LIN {X 0,Y 516.423,Z 190.622,A -85,B 0,C 180,E1 -4930.11,E2 -4930.11} C_VEL
LIN {X 0,Y 516.366,Z 194.851,A -85,B 0,C 180,E1 -4932.577,E2 -4932.577} C_VEL
LIN {X 0,Y 516.329,Z 197.599,A -85,B 0,C 180,E1 -4934.178,E2 -4934.178} C_VEL
LIN {X 0,Y 518.484,Z 209.749,A -85,B 0,C 180,E1 -4934.55,E2 -4934.55} C_VEL
LIN {X 0,Y 518.248,Z 221.683,A -85,B 0,C 180,E1 -4934.993,E2 -4934.993} C_VEL
LIN {X 0,Y 517.972,Z 233.125,A -85,B 0,C 180,E1 -4935.563,E2 -4935.563} C_VEL
LIN {X 0,Y 517.62,Z 243.966,A -85,B 0,C 180,E1 -4936.255,E2 -4936.255} C_VEL
LIN {X 0,Y 517.384,Z 254.996,A -85,B 0,C 180,E1 -4937.148,E2 -4937.148} C_VEL
LIN {X 0,Y 517.083,Z 264.736,A -85,B 0,C 180,E1 -4938.127,E2 -4938.127} C_VEL
LIN {X 0,Y 516.875,Z 273.613,A -85,B 0,C 180,E1 -4939.225,E2 -4939.225} C_VEL
LIN {X 0,Y 516.618,Z 281.309,A -85,B 0,C 180,E1 -4940.407,E2 -4940.407} C_VEL
LIN {X 0,Y 516.474,Z 288.372,A -85,B 0,C 180,E1 -4941.786,E2 -4941.786} C_VEL
LIN {X 0,Y 516.395,Z 293.063,A -85,B 0,C 180,E1 -4942.964,E2 -4942.964} C_VEL
LIN {X 0,Y 516.305,Z 296.646,A -85,B 0,C 180,E1 -4944.14,E2 -4944.14} C_VEL
LIN {X 0,Y 516.227,Z 299.218,A -85,B 0,C 180,E1 -4945.314,E2 -4945.314} C_VEL
LIN {X 0,Y 516.326,Z 300.425,A -85,B 0,C 180,E1 -4946.097,E2 -4946.097} C_VEL
LIN {X 0,Y 516.274,Z 301.209,A -85,B 0,C 180,E1 -4946.878,E2 -4946.878} C_VEL
LIN {X 0,Y 516.26,Z 301.586,A -85,B 0,C 180,E1 -4947.659,E2 -4947.659} C_VEL
LIN {X 0,Y 516.162,Z 301.206,A -85,B 0,C 180,E1 -4949.219,E2 -4949.219} C_VEL
LIN {X 0,Y 516.162,Z 300.418,A -85,B 0,C 180,E1 -4949.999,E2 -4949.999} C_VEL
LIN {X 0,Y 516.222,Z 297.602,A -85,B 0,C 180,E1 -4951.56,E2 -4951.56} C_VEL
LIN {X 0,Y 516.35,Z 294.377,A -85,B 0,C 180,E1 -4952.73,E2 -4952.73} C_VEL
LIN {X 0,Y 516.429,Z 290.102,A -85,B 0,C 180,E1 -4953.901,E2 -4953.901} C_VEL
LIN {X 0,Y 516.634,Z 284.648,A -85,B 0,C 180,E1 -4955.072,E2 -4955.072} C_VEL
LIN {X 0,Y 516.739,Z 277.853,A -85,B 0,C 180,E1 -4956.245,E2 -4956.245} C_VEL
LIN {X 0,Y 516.941,Z 269.359,A -85,B 0,C 180,E1 -4957.42,E2 -4957.42} C_VEL
LIN {X 0,Y 517.257,Z 260.641,A -85,B 0,C 180,E1 -4958.398,E2 -4958.398} C_VEL
LIN {X 0,Y 517.567,Z 249.918,A -85,B 0,C 180,E1 -4959.377,E2 -4959.377} C_VEL
LIN {X 0,Y 517.823,Z 239.153,A -85,B 0,C 180,E1 -4960.161,E2 -4960.161} C_VEL
LIN {X 0,Y 518.117,Z 227.088,A -85,B 0,C 180,E1 -4960.847,E2 -4960.847} C_VEL
LIN {X 0,Y 518.374,Z 215.239,A -85,B 0,C 180,E1 -4961.355,E2 -4961.355} C_VEL
LIN {X 0,Y 518.352,Z 208.104,A -85,B 0,C 180,E1 -4961.595,E2 -4961.595} C_VEL
LIN {X 0,Y 516.358,Z 197.517,A -85,B 0,C 180,E1 -4961.93,E2 -4961.93} C_VEL
LIN {X 0,Y 516.455,Z 192.31,A -85,B 0,C 180,E1 -4964.983,E2 -4964.983} C_VEL
LIN {X 0,Y 516.434,Z 186.816,A -85,B 0,C 180,E1 -4968.238,E2 -4968.238} C_VEL
LIN {X 0,Y 516.53,Z 182.754,A -85,B 0,C 180,E1 -4970.715,E2 -4970.715} C_VEL
LIN {X 0,Y 516.546,Z 178.687,A -85,B 0,C 180,E1 -4973.237,E2 -4973.237} C_VEL
LIN {X 0,Y 516.626,Z 174.098,A -85,B 0,C 180,E1 -4976.123,E2 -4976.123} C_VEL
LIN {X 0,Y 516.738,Z 169.128,A -85,B 0,C 180,E1 -4979.313,E2 -4979.313} C_VEL
LIN {X 0,Y 516.758,Z 164.99,A -85,B 0,C 180,E1 -4982.03,E2 -4982.03} C_VEL
LIN {X 0,Y 516.75,Z 163.594,A -85,B 0,C 180,E1 -4982.954,E2 -4982.954} C_VEL
LIN {X 0,Y 516.827,Z 163.108,A -85,B 0,C 180,E1 -4983.952,E2 -4983.952} C_VEL
LIN {X 0,Y 516.84,Z 163.107,A -85,B 0,C 180,E1 -4986.745,E2 -4986.745} C_VEL
LIN {X 0,Y 516.867,Z 163.102,A -85,B 0,C 180,E1 -4989.719,E2 -4989.719} C_VEL
LIN {X 0,Y 516.89,Z 163.097,A -85,B 0,C 180,E1 -4992.758,E2 -4992.758} C_VEL
LIN {X 0,Y 516.904,Z 163.097,A -85,B 0,C 180,E1 -4995.007,E2 -4995.007} C_VEL
LIN {X 0,Y 516.908,Z 163.094,A -85,B 0,C 180,E1 -4998.394,E2 -4998.394} C_VEL
LIN {X 0,Y 516.862,Z 163.101,A -85,B 0,C 180,E1 -5001.282,E2 -5001.282} C_VEL
LIN {X 0,Y 516.85,Z 163.106,A -85,B 0,C 180,E1 -5004.217,E2 -5004.217} C_VEL
LIN {X 0,Y 516.871,Z 163.101,A -85,B 0,C 180,E1 -5007.051,E2 -5007.051} C_VEL
LIN {X 0,Y 516.874,Z 163.101,A -85,B 0,C 180,E1 -5009.795,E2 -5009.795} C_VEL
LIN {X 0,Y 516.904,Z 163.097,A -85,B 0,C 180,E1 -5012.466,E2 -5012.466} C_VEL
LIN {X 0,Y 516.913,Z 163.095,A -85,B 0,C 180,E1 -5015.072,E2 -5015.072} C_VEL
LIN {X 0,Y 516.879,Z 163.099,A -85,B 0,C 180,E1 -5017.622,E2 -5017.622} C_VEL
LIN {X 0,Y 516.896,Z 163.1,A -85,B 0,C 180,E1 -5020.128,E2 -5020.128} C_VEL
LIN {X 0,Y 516.898,Z 163.097,A -85,B 0,C 180,E1 -5022.595,E2 -5022.595} C_VEL
LIN {X 0,Y 516.885,Z 163.098,A -85,B 0,C 180,E1 -5025.833,E2 -5025.833} C_VEL
LIN {X 0,Y 516.994,Z 163.087,A -85,B 0,C 180,E1 -5028.234,E2 -5028.234} C_VEL
LIN {X 0,Y 516.947,Z 163.089,A -85,B 0,C 180,E1 -5031.399,E2 -5031.399} C_VEL
LIN {X 0,Y 517.005,Z 163.087,A -85,B 0,C 180,E1 -5033.757,E2 -5033.757} C_VEL
LIN {X 0,Y 516.982,Z 163.087,A -85,B 0,C 180,E1 -5036.883,E2 -5036.883} C_VEL
LIN {X 0,Y 517.039,Z 163.079,A -85,B 0,C 180,E1 -5040,E2 -5040} C_VEL
LIN {X 0,Y 517.014,Z 163.083,A -85,B 0,C 180,E1 -5043.117,E2 -5043.117} C_VEL
LIN {X 0,Y 516.998,Z 163.086,A -85,B 0,C 180,E1 -5046.243,E2 -5046.243} C_VEL
LIN {X 0,Y 516.946,Z 163.089,A -85,B 0,C 180,E1 -5048.601,E2 -5048.601} C_VEL
LIN {X 0,Y 516.965,Z 163.088,A -85,B 0,C 180,E1 -5051.835,E2 -5051.835} C_VEL
LIN {X 0,Y 516.908,Z 163.097,A -85,B 0,C 180,E1 -5055.148,E2 -5055.148} C_VEL
LIN {X 0,Y 516.889,Z 163.101,A -85,B 0,C 180,E1 -5058.223,E2 -5058.223} C_VEL
LIN {X 0,Y 516.882,Z 163.099,A -85,B 0,C 180,E1 -5060.703,E2 -5060.703} C_VEL
LIN {X 0,Y 516.877,Z 163.103,A -85,B 0,C 180,E1 -5063.223,E2 -5063.223} C_VEL
LIN {X 0,Y 516.918,Z 163.093,A -85,B 0,C 180,E1 -5066.2,E2 -5066.2} C_VEL
LIN {X 0,Y 516.912,Z 163.094,A -85,B 0,C 180,E1 -5069.305,E2 -5069.305} C_VEL
LIN {X 0,Y 516.87,Z 163.102,A -85,B 0,C 180,E1 -5072.546,E2 -5072.546} C_VEL
LIN {X 0,Y 516.852,Z 163.105,A -85,B 0,C 180,E1 -5075.334,E2 -5075.334} C_VEL
LIN {X 0,Y 516.856,Z 163.103,A -85,B 0,C 180,E1 -5077.946,E2 -5077.946} C_VEL
LIN {X 0,Y 516.885,Z 163.103,A -85,B 0,C 180,E1 -5080.742,E2 -5080.742} C_VEL
LIN {X 0,Y 516.861,Z 163.101,A -85,B 0,C 180,E1 -5083.906,E2 -5083.906} C_VEL
LIN {X 0,Y 516.863,Z 163.106,A -85,B 0,C 180,E1 -5086.109,E2 -5086.109} C_VEL
LIN {X 0,Y 516.899,Z 163.1,A -85,B 0,C 180,E1 -5088.401,E2 -5088.401} C_VEL
LIN {X 0,Y 516.862,Z 163.107,A -85,B 0,C 180,E1 -5091.286,E2 -5091.286} C_VEL
LIN {X 0,Y 516.902,Z 163.236,A -85,B 0,C 180,E1 -5092.527,E2 -5092.527} C_VEL
LIN {X 0,Y 517.536,Z 167.733,A -85,B 0,C 180,E1 -5094.566,E2 -5094.566} C_VEL
LIN {X 0,Y 517.365,Z 174.379,A -85,B 0,C 180,E1 -5097.376,E2 -5097.376} C_VEL
LIN {X 0,Y 517.206,Z 181.852,A -85,B 0,C 180,E1 -5100.419,E2 -5100.419} C_VEL
LIN {X 0,Y 517,Z 190.448,A -85,B 0,C 180,E1 -5103.792,E2 -5103.792} C_VEL
LIN {X 0,Y 516.782,Z 198.275,A -85,B 0,C 180,E1 -5106.775,E2 -5106.775} C_VEL
LIN {X 0,Y 516.657,Z 206.41,A -85,B 0,C 180,E1 -5109.818,E2 -5109.818} C_VEL
LIN {X 0,Y 516.526,Z 213.919,A -85,B 0,C 180,E1 -5112.584,E2 -5112.584} C_VEL
LIN {X 0,Y 516.474,Z 221.738,A -85,B 0,C 180,E1 -5115.437,E2 -5115.437} C_VEL
LIN {X 0,Y 516.467,Z 223.583,A -85,B 0,C 180,E1 -5116.099,E2 -5116.099} C_VEL
LIN {X 0,Y 518.43,Z 237.052,A -85,B 0,C 180,E1 -5116.478,E2 -5116.478} C_VEL
LIN {X 0,Y 518.121,Z 250.37,A -85,B 0,C 180,E1 -5116.969,E2 -5116.969} C_VEL
LIN {X 0,Y 517.817,Z 263.139,A -85,B 0,C 180,E1 -5117.619,E2 -5117.619} C_VEL
LIN {X 0,Y 517.542,Z 274.076,A -85,B 0,C 180,E1 -5118.348,E2 -5118.348} C_VEL
LIN {X 0,Y 517.25,Z 284.743,A -85,B 0,C 180,E1 -5119.234,E2 -5119.234} C_VEL
LIN {X 0,Y 516.944,Z 294.354,A -85,B 0,C 180,E1 -5120.217,E2 -5120.217} C_VEL
LIN {X 0,Y 516.735,Z 302.234,A -85,B 0,C 180,E1 -5121.2,E2 -5121.2} C_VEL
LIN {X 0,Y 516.539,Z 309.929,A -85,B 0,C 180,E1 -5122.378,E2 -5122.378} C_VEL
LIN {X 0,Y 516.393,Z 317.023,A -85,B 0,C 180,E1 -5123.75,E2 -5123.75} C_VEL
LIN {X 0,Y 516.313,Z 321.743,A -85,B 0,C 180,E1 -5124.925,E2 -5124.925} C_VEL
LIN {X 0,Y 516.352,Z 325.351,A -85,B 0,C 180,E1 -5126.099,E2 -5126.099} C_VEL
LIN {X 0,Y 516.282,Z 327.209,A -85,B 0,C 180,E1 -5126.879,E2 -5126.879} C_VEL
LIN {X 0,Y 516.261,Z 328.603,A -85,B 0,C 180,E1 -5127.66,E2 -5127.66} C_VEL
LIN {X 0,Y 516.16,Z 330.203,A -85,B 0,C 180,E1 -5129.22,E2 -5129.22} C_VEL
LIN {X 0,Y 516.156,Z 330.418,A -85,B 0,C 180,E1 -5130.001,E2 -5130.001} C_VEL
LIN {X 0,Y 516.192,Z 329.596,A -85,B 0,C 180,E1 -5131.561,E2 -5131.561} C_VEL
LIN {X 0,Y 516.261,Z 328.603,A -85,B 0,C 180,E1 -5132.341,E2 -5132.341} C_VEL
LIN {X 0,Y 516.282,Z 327.209,A -85,B 0,C 180,E1 -5133.122,E2 -5133.122} C_VEL
LIN {X 0,Y 516.312,Z 324.275,A -85,B 0,C 180,E1 -5134.294,E2 -5134.294} C_VEL
LIN {X 0,Y 516.375,Z 320.304,A -85,B 0,C 180,E1 -5135.467,E2 -5135.467} C_VEL
LIN {X 0,Y 516.478,Z 314.404,A -85,B 0,C 180,E1 -5136.798,E2 -5136.798} C_VEL
LIN {X 0,Y 516.604,Z 307.521,A -85,B 0,C 180,E1 -5138.016,E2 -5138.016} C_VEL
LIN {X 0,Y 516.822,Z 299.24,A -85,B 0,C 180,E1 -5139.194,E2 -5139.194} C_VEL
LIN {X 0,Y 517.037,Z 290.752,A -85,B 0,C 180,E1 -5140.178,E2 -5140.178} C_VEL
LIN {X 0,Y 517.347,Z 280.265,A -85,B 0,C 180,E1 -5141.162,E2 -5141.162} C_VEL
LIN {X 0,Y 517.651,Z 269.287,A -85,B 0,C 180,E1 -5141.991,E2 -5141.991} C_VEL
LIN {X 0,Y 517.937,Z 258.519,A -85,B 0,C 180,E1 -5142.638,E2 -5142.638} C_VEL
LIN {X 0,Y 518.253,Z 246.86,A -85,B 0,C 180,E1 -5143.179,E2 -5143.179} C_VEL
LIN {X 0,Y 518.238,Z 235.249,A -85,B 0,C 180,E1 -5143.578,E2 -5143.578} C_VEL
LIN {X 0,Y 516.453,Z 223.564,A -85,B 0,C 180,E1 -5143.902,E2 -5143.902} C_VEL
LIN {X 0,Y 516.524,Z 214.964,A -85,B 0,C 180,E1 -5147.009,E2 -5147.009} C_VEL
LIN {X 0,Y 516.639,Z 207.215,A -85,B 0,C 180,E1 -5149.881,E2 -5149.881} C_VEL
LIN {X 0,Y 516.765,Z 199.392,A -85,B 0,C 180,E1 -5152.804,E2 -5152.804} C_VEL
LIN {X 0,Y 516.919,Z 192.705,A -85,B 0,C 180,E1 -5155.357,E2 -5155.357} C_VEL
LIN {X 0,Y 517.152,Z 184.948,A -85,B 0,C 180,E1 -5158.4,E2 -5158.4} C_VEL
LIN {X 0,Y 517.347,Z 177.234,A -85,B 0,C 180,E1 -5161.532,E2 -5161.532} C_VEL
LIN {X 0,Y 517.478,Z 171.26,A -85,B 0,C 180,E1 -5164.059,E2 -5164.059} C_VEL
LIN {X 0,Y 517.526,Z 167.439,A -85,B 0,C 180,E1 -5165.726,E2 -5165.726} C_VEL
LIN {X 0,Y 516.87,Z 163.106,A -85,B 0,C 180,E1 -5167.799,E2 -5167.799} C_VEL
LIN {X 0,Y 516.874,Z 163.101,A -85,B 0,C 180,E1 -5170.74,E2 -5170.74} C_VEL
LIN {X 0,Y 516.893,Z 163.097,A -85,B 0,C 180,E1 -5172.827,E2 -5172.827} C_VEL
LIN {X 0,Y 516.909,Z 163.099,A -85,B 0,C 180,E1 -5175.008,E2 -5175.008} C_VEL
LIN {X 0,Y 516.896,Z 163.1,A -85,B 0,C 180,E1 -5178.397,E2 -5178.397} C_VEL
LIN {X 0,Y 516.862,Z 163.102,A -85,B 0,C 180,E1 -5181.282,E2 -5181.282} C_VEL
LIN {X 0,Y 516.872,Z 163.099,A -85,B 0,C 180,E1 -5184.22,E2 -5184.22} C_VEL
LIN {X 0,Y 516.877,Z 163.104,A -85,B 0,C 180,E1 -5187.052,E2 -5187.052} C_VEL
LIN {X 0,Y 516.878,Z 163.1,A -85,B 0,C 180,E1 -5189.795,E2 -5189.795} C_VEL
LIN {X 0,Y 516.903,Z 163.098,A -85,B 0,C 180,E1 -5192.466,E2 -5192.466} C_VEL
LIN {X 0,Y 516.897,Z 163.099,A -85,B 0,C 180,E1 -5195.071,E2 -5195.071} C_VEL
LIN {X 0,Y 516.887,Z 163.097,A -85,B 0,C 180,E1 -5197.622,E2 -5197.622} C_VEL
LIN {X 0,Y 516.906,Z 163.097,A -85,B 0,C 180,E1 -5200.129,E2 -5200.129} C_VEL
LIN {X 0,Y 516.915,Z 163.097,A -85,B 0,C 180,E1 -5202.596,E2 -5202.596} C_VEL
LIN {X 0,Y 516.911,Z 163.097,A -85,B 0,C 180,E1 -5205.029,E2 -5205.029} C_VEL
LIN {X 0,Y 516.975,Z 163.087,A -85,B 0,C 180,E1 -5208.234,E2 -5208.234} C_VEL
LIN {X 0,Y 516.949,Z 163.089,A -85,B 0,C 180,E1 -5211.399,E2 -5211.399} C_VEL
LIN {X 0,Y 517.014,Z 163.084,A -85,B 0,C 180,E1 -5213.757,E2 -5213.757} C_VEL
LIN {X 0,Y 516.988,Z 163.088,A -85,B 0,C 180,E1 -5216.883,E2 -5216.883} C_VEL
LIN {X 0,Y 517.048,Z 163.078,A -85,B 0,C 180,E1 -5220,E2 -5220} C_VEL
LIN {X 0,Y 517.022,Z 163.08,A -85,B 0,C 180,E1 -5223.117,E2 -5223.117} C_VEL
LIN {X 0,Y 516.99,Z 163.086,A -85,B 0,C 180,E1 -5226.244,E2 -5226.244} C_VEL
LIN {X 0,Y 516.93,Z 163.096,A -85,B 0,C 180,E1 -5229.39,E2 -5229.39} C_VEL
LIN {X 0,Y 516.924,Z 163.094,A -85,B 0,C 180,E1 -5231.809,E2 -5231.809} C_VEL
LIN {X 0,Y 516.915,Z 163.094,A -85,B 0,C 180,E1 -5235.147,E2 -5235.147} C_VEL
LIN {X 0,Y 516.905,Z 163.095,A -85,B 0,C 180,E1 -5238.223,E2 -5238.223} C_VEL
LIN {X 0,Y 516.89,Z 163.1,A -85,B 0,C 180,E1 -5240.703,E2 -5240.703} C_VEL
LIN {X 0,Y 516.856,Z 163.103,A -85,B 0,C 180,E1 -5243.225,E2 -5243.225} C_VEL
LIN {X 0,Y 516.921,Z 163.096,A -85,B 0,C 180,E1 -5246.198,E2 -5246.198} C_VEL
LIN {X 0,Y 516.914,Z 163.1,A -85,B 0,C 180,E1 -5249.305,E2 -5249.305} C_VEL
LIN {X 0,Y 516.881,Z 163.102,A -85,B 0,C 180,E1 -5252.546,E2 -5252.546} C_VEL
LIN {X 0,Y 516.86,Z 163.102,A -85,B 0,C 180,E1 -5255.334,E2 -5255.334} C_VEL
LIN {X 0,Y 516.862,Z 163.104,A -85,B 0,C 180,E1 -5257.945,E2 -5257.945} C_VEL
LIN {X 0,Y 516.871,Z 163.102,A -85,B 0,C 180,E1 -5260.743,E2 -5260.743} C_VEL
LIN {X 0,Y 516.871,Z 163.104,A -85,B 0,C 180,E1 -5262.833,E2 -5262.833} C_VEL
LIN {X 0,Y 516.911,Z 163.095,A -85,B 0,C 180,E1 -5265.012,E2 -5265.012} C_VEL
LIN {X 0,Y 516.904,Z 163.097,A -85,B 0,C 180,E1 -5268.401,E2 -5268.401} C_VEL
LIN {X 0,Y 516.851,Z 163.103,A -85,B 0,C 180,E1 -5270.332,E2 -5270.332} C_VEL
LIN {X 0,Y 516.18,Z 163.195,A -85,B 0,C 180,E1 -5270.982,E2 -5270.982} C_VEL
LIN {X 0,Y 513.3,Z 163.735,A -85,B 0,C 180,E1 -5272.035,E2 -5272.035} C_VEL
LIN {X 0,Y 510.862,Z 164.526,A -85,B 0,C 180,E1 -5272.88,E2 -5272.88} C_VEL
LIN {X 0,Y 509.812,Z 165.338,A -85,B 0,C 180,E1 -5273.531,E2 -5273.531} C_VEL
LIN {X 0,Y 509.725,Z 165.651,A -85,B 0,C 180,E1 -5273.75,E2 -5273.75} C_VEL
LIN {X 0,Y 509.698,Z 169.763,A -85,B 0,C 180,E1 -5276.529,E2 -5276.529} C_VEL
LIN {X 0,Y 509.59,Z 173.994,A -85,B 0,C 180,E1 -5279.319,E2 -5279.319} C_VEL
LIN {X 0,Y 509.548,Z 178.187,A -85,B 0,C 180,E1 -5282.036,E2 -5282.036} C_VEL
LIN {X 0,Y 509.474,Z 182.359,A -85,B 0,C 180,E1 -5284.684,E2 -5284.684} C_VEL
LIN {X 0,Y 509.377,Z 187.013,A -85,B 0,C 180,E1 -5287.582,E2 -5287.582} C_VEL
LIN {X 0,Y 509.3,Z 192.127,A -85,B 0,C 180,E1 -5290.66,E2 -5290.66} C_VEL
LIN {X 0,Y 509.246,Z 196.339,A -85,B 0,C 180,E1 -5293.154,E2 -5293.154} C_VEL
LIN {X 0,Y 509.265,Z 197.751,A -85,B 0,C 180,E1 -5293.979,E2 -5293.979} C_VEL
LIN {X 0,Y 511.578,Z 210.681,A -85,B 0,C 180,E1 -5294.389,E2 -5294.389} C_VEL
LIN {X 0,Y 511.304,Z 222.986,A -85,B 0,C 180,E1 -5294.862,E2 -5294.862} C_VEL
LIN {X 0,Y 511.005,Z 234.608,A -85,B 0,C 180,E1 -5295.464,E2 -5295.464} C_VEL
LIN {X 0,Y 510.587,Z 246.462,A -85,B 0,C 180,E1 -5296.265,E2 -5296.265} C_VEL
LIN {X 0,Y 510.36,Z 257.042,A -85,B 0,C 180,E1 -5297.171,E2 -5297.171} C_VEL
LIN {X 0,Y 510.011,Z 266.994,A -85,B 0,C 180,E1 -5298.224,E2 -5298.224} C_VEL
LIN {X 0,Y 509.83,Z 275.011,A -85,B 0,C 180,E1 -5299.275,E2 -5299.275} C_VEL
LIN {X 0,Y 509.571,Z 282.468,A -85,B 0,C 180,E1 -5300.474,E2 -5300.474} C_VEL
LIN {X 0,Y 509.401,Z 288.446,A -85,B 0,C 180,E1 -5301.671,E2 -5301.671} C_VEL
LIN {X 0,Y 509.321,Z 293.164,A -85,B 0,C 180,E1 -5302.866,E2 -5302.866} C_VEL
LIN {X 0,Y 509.232,Z 296.77,A -85,B 0,C 180,E1 -5304.059,E2 -5304.059} C_VEL
LIN {X 0,Y 509.145,Z 299.366,A -85,B 0,C 180,E1 -5305.249,E2 -5305.249} C_VEL
LIN {X 0,Y 509.232,Z 300.585,A -85,B 0,C 180,E1 -5306.043,E2 -5306.043} C_VEL
LIN {X 0,Y 509.192,Z 301.39,A -85,B 0,C 180,E1 -5306.835,E2 -5306.835} C_VEL
LIN {X 0,Y 509.189,Z 301.778,A -85,B 0,C 180,E1 -5307.627,E2 -5307.627} C_VEL
LIN {X 0,Y 509.075,Z 301.42,A -85,B 0,C 180,E1 -5309.209,E2 -5309.209} C_VEL
LIN {X 0,Y 509.073,Z 300.653,A -85,B 0,C 180,E1 -5309.999,E2 -5309.999} C_VEL
LIN {X 0,Y 509.143,Z 297.86,A -85,B 0,C 180,E1 -5311.581,E2 -5311.581} C_VEL
LIN {X 0,Y 509.282,Z 294.659,A -85,B 0,C 180,E1 -5312.768,E2 -5312.768} C_VEL
LIN {X 0,Y 509.365,Z 290.409,A -85,B 0,C 180,E1 -5313.955,E2 -5313.955} C_VEL
LIN {X 0,Y 509.58,Z 284.983,A -85,B 0,C 180,E1 -5315.142,E2 -5315.142} C_VEL
LIN {X 0,Y 509.709,Z 278.218,A -85,B 0,C 180,E1 -5316.332,E2 -5316.332} C_VEL
LIN {X 0,Y 509.923,Z 269.779,A -85,B 0,C 180,E1 -5317.522,E2 -5317.522} C_VEL
LIN {X 0,Y 510.267,Z 261.104,A -85,B 0,C 180,E1 -5318.513,E2 -5318.513} C_VEL
LIN {X 0,Y 510.587,Z 250.436,A -85,B 0,C 180,E1 -5319.506,E2 -5319.506} C_VEL
LIN {X 0,Y 510.863,Z 239.78,A -85,B 0,C 180,E1 -5320.301,E2 -5320.301} C_VEL
LIN {X 0,Y 511.184,Z 227.828,A -85,B 0,C 180,E1 -5320.996,E2 -5320.996} C_VEL
LIN {X 0,Y 511.49,Z 215.533,A -85,B 0,C 180,E1 -5321.534,E2 -5321.534} C_VEL
LIN {X 0,Y 511.357,Z 208.331,A -85,B 0,C 180,E1 -5321.783,E2 -5321.783} C_VEL
LIN {X 0,Y 509.266,Z 197.718,A -85,B 0,C 180,E1 -5322.127,E2 -5322.127} C_VEL
LIN {X 0,Y 509.367,Z 192.502,A -85,B 0,C 180,E1 -5325.196,E2 -5325.196} C_VEL
LIN {X 0,Y 509.385,Z 188.102,A -85,B 0,C 180,E1 -5327.824,E2 -5327.824} C_VEL
LIN {X 0,Y 509.46,Z 182.923,A -85,B 0,C 180,E1 -5331.016,E2 -5331.016} C_VEL
LIN {X 0,Y 509.482,Z 178.842,A -85,B 0,C 180,E1 -5333.578,E2 -5333.578} C_VEL
LIN {X 0,Y 509.575,Z 174.566,A -85,B 0,C 180,E1 -5336.301,E2 -5336.301} C_VEL
LIN {X 0,Y 509.636,Z 170.633,A -85,B 0,C 180,E1 -5338.856,E2 -5338.856} C_VEL
LIN {X 0,Y 509.719,Z 166.487,A -85,B 0,C 180,E1 -5341.594,E2 -5341.594} C_VEL
LIN {X 0,Y 509.709,Z 163.998,A -85,B 0,C 180,E1 -5343.469,E2 -5343.469} C_VEL
LIN {X 0,Y 509.809,Z 163.98,A -85,B 0,C 180,E1 -5345.575,E2 -5345.575} C_VEL
LIN {X 0,Y 509.835,Z 163.979,A -85,B 0,C 180,E1 -5348.335,E2 -5348.335} C_VEL
LIN {X 0,Y 509.843,Z 163.976,A -85,B 0,C 180,E1 -5351.422,E2 -5351.422} C_VEL
LIN {X 0,Y 509.839,Z 163.975,A -85,B 0,C 180,E1 -5354.665,E2 -5354.665} C_VEL
LIN {X 0,Y 509.866,Z 163.971,A -85,B 0,C 180,E1 -5358.097,E2 -5358.097} C_VEL
LIN {X 0,Y 509.837,Z 163.98,A -85,B 0,C 180,E1 -5360.646,E2 -5360.646} C_VEL
LIN {X 0,Y 509.801,Z 163.982,A -85,B 0,C 180,E1 -5363.644,E2 -5363.644} C_VEL
LIN {X 0,Y 509.835,Z 163.977,A -85,B 0,C 180,E1 -5366.537,E2 -5366.537} C_VEL
LIN {X 0,Y 509.823,Z 163.982,A -85,B 0,C 180,E1 -5369.332,E2 -5369.332} C_VEL
LIN {X 0,Y 509.869,Z 163.971,A -85,B 0,C 180,E1 -5372.053,E2 -5372.053} C_VEL
LIN {X 0,Y 509.869,Z 163.976,A -85,B 0,C 180,E1 -5374.703,E2 -5374.703} C_VEL
LIN {X 0,Y 509.851,Z 163.974,A -85,B 0,C 180,E1 -5377.44,E2 -5377.44} C_VEL
LIN {X 0,Y 509.881,Z 163.974,A -85,B 0,C 180,E1 -5379.843,E2 -5379.843} C_VEL
LIN {X 0,Y 509.857,Z 163.977,A -85,B 0,C 180,E1 -5383.174,E2 -5383.174} C_VEL
LIN {X 0,Y 509.847,Z 163.976,A -85,B 0,C 180,E1 -5385.633,E2 -5385.633} C_VEL
LIN {X 0,Y 509.925,Z 163.967,A -85,B 0,C 180,E1 -5388.875,E2 -5388.875} C_VEL
LIN {X 0,Y 509.948,Z 163.968,A -85,B 0,C 180,E1 -5392.078,E2 -5392.078} C_VEL
LIN {X 0,Y 509.988,Z 163.957,A -85,B 0,C 180,E1 -5394.464,E2 -5394.464} C_VEL
LIN {X 0,Y 510.015,Z 163.957,A -85,B 0,C 180,E1 -5397.631,E2 -5397.631} C_VEL
LIN {X 0,Y 510.029,Z 163.955,A -85,B 0,C 180,E1 -5400.789,E2 -5400.789} C_VEL
LIN {X 0,Y 509.954,Z 163.962,A -85,B 0,C 180,E1 -5403.16,E2 -5403.16} C_VEL
LIN {X 0,Y 509.962,Z 163.962,A -85,B 0,C 180,E1 -5406.33,E2 -5406.33} C_VEL
LIN {X 0,Y 509.919,Z 163.964,A -85,B 0,C 180,E1 -5408.72,E2 -5408.72} C_VEL
LIN {X 0,Y 509.916,Z 163.965,A -85,B 0,C 180,E1 -5411.931,E2 -5411.931} C_VEL
LIN {X 0,Y 509.856,Z 163.975,A -85,B 0,C 180,E1 -5415.243,E2 -5415.243} C_VEL
LIN {X 0,Y 509.851,Z 163.978,A -85,B 0,C 180,E1 -5418.002,E2 -5418.002} C_VEL
LIN {X 0,Y 509.826,Z 163.978,A -85,B 0,C 180,E1 -5421.003,E2 -5421.003} C_VEL
LIN {X 0,Y 509.836,Z 163.979,A -85,B 0,C 180,E1 -5423.563,E2 -5423.563} C_VEL
LIN {X 0,Y 509.887,Z 163.969,A -85,B 0,C 180,E1 -5426.382,E2 -5426.382} C_VEL
LIN {X 0,Y 509.86,Z 163.977,A -85,B 0,C 180,E1 -5428.845,E2 -5428.845} C_VEL
LIN {X 0,Y 509.796,Z 163.982,A -85,B 0,C 180,E1 -5431.592,E2 -5431.592} C_VEL
LIN {X 0,Y 509.823,Z 163.979,A -85,B 0,C 180,E1 -5434.416,E2 -5434.416} C_VEL
LIN {X 0,Y 509.793,Z 163.985,A -85,B 0,C 180,E1 -5437.343,E2 -5437.343} C_VEL
LIN {X 0,Y 509.839,Z 163.977,A -85,B 0,C 180,E1 -5440.382,E2 -5440.382} C_VEL
LIN {X 0,Y 509.819,Z 163.979,A -85,B 0,C 180,E1 -5443.067,E2 -5443.067} C_VEL
LIN {X 0,Y 509.811,Z 163.981,A -85,B 0,C 180,E1 -5445.795,E2 -5445.795} C_VEL
LIN {X 0,Y 509.841,Z 163.979,A -85,B 0,C 180,E1 -5448.577,E2 -5448.577} C_VEL
LIN {X 0,Y 509.834,Z 163.981,A -85,B 0,C 180,E1 -5451.789,E2 -5451.789} C_VEL
LIN {X 0,Y 509.839,Z 164.11,A -85,B 0,C 180,E1 -5452.354,E2 -5452.354} C_VEL
LIN {X 0,Y 510.537,Z 169.183,A -85,B 0,C 180,E1 -5454.682,E2 -5454.682} C_VEL
LIN {X 0,Y 510.325,Z 175.809,A -85,B 0,C 180,E1 -5457.517,E2 -5457.517} C_VEL
LIN {X 0,Y 510.172,Z 183.589,A -85,B 0,C 180,E1 -5460.726,E2 -5460.726} C_VEL
LIN {X 0,Y 509.897,Z 192.538,A -85,B 0,C 180,E1 -5464.27,E2 -5464.27} C_VEL
LIN {X 0,Y 509.71,Z 200.377,A -85,B 0,C 180,E1 -5467.292,E2 -5467.292} C_VEL
LIN {X 0,Y 509.593,Z 207.09,A -85,B 0,C 180,E1 -5469.833,E2 -5469.833} C_VEL
LIN {X 0,Y 509.458,Z 214.878,A -85,B 0,C 180,E1 -5472.749,E2 -5472.749} C_VEL
LIN {X 0,Y 509.367,Z 223.383,A -85,B 0,C 180,E1 -5475.902,E2 -5475.902} C_VEL
LIN {X 0,Y 511.464,Z 237.235,A -85,B 0,C 180,E1 -5476.303,E2 -5476.303} C_VEL
LIN {X 0,Y 511.211,Z 250.172,A -85,B 0,C 180,E1 -5476.789,E2 -5476.789} C_VEL
LIN {X 0,Y 510.895,Z 261.567,A -85,B 0,C 180,E1 -5477.369,E2 -5477.369} C_VEL
LIN {X 0,Y 510.589,Z 272.564,A -85,B 0,C 180,E1 -5478.086,E2 -5478.086} C_VEL
LIN {X 0,Y 510.284,Z 283.472,A -85,B 0,C 180,E1 -5478.985,E2 -5478.985} C_VEL
LIN {X 0,Y 509.951,Z 292.367,A -85,B 0,C 180,E1 -5479.881,E2 -5479.881} C_VEL
LIN {X 0,Y 509.684,Z 302.035,A -85,B 0,C 180,E1 -5481.077,E2 -5481.077} C_VEL
LIN {X 0,Y 509.476,Z 309.731,A -85,B 0,C 180,E1 -5482.272,E2 -5482.272} C_VEL
LIN {X 0,Y 509.307,Z 316.825,A -85,B 0,C 180,E1 -5483.663,E2 -5483.663} C_VEL
LIN {X 0,Y 509.246,Z 321.546,A -85,B 0,C 180,E1 -5484.854,E2 -5484.854} C_VEL
LIN {X 0,Y 509.245,Z 325.153,A -85,B 0,C 180,E1 -5486.044,E2 -5486.044} C_VEL
LIN {X 0,Y 509.2,Z 327.012,A -85,B 0,C 180,E1 -5486.836,E2 -5486.836} C_VEL
LIN {X 0,Y 509.19,Z 328.406,A -85,B 0,C 180,E1 -5487.628,E2 -5487.628} C_VEL
LIN {X 0,Y 509.074,Z 330.005,A -85,B 0,C 180,E1 -5489.21,E2 -5489.21} C_VEL
LIN {X 0,Y 509.067,Z 330.221,A -85,B 0,C 180,E1 -5490.001,E2 -5490.001} C_VEL
LIN {X 0,Y 509.112,Z 329.399,A -85,B 0,C 180,E1 -5491.582,E2 -5491.582} C_VEL
LIN {X 0,Y 509.19,Z 328.406,A -85,B 0,C 180,E1 -5492.373,E2 -5492.373} C_VEL
LIN {X 0,Y 509.2,Z 327.011,A -85,B 0,C 180,E1 -5493.165,E2 -5493.165} C_VEL
LIN {X 0,Y 509.204,Z 324.076,A -85,B 0,C 180,E1 -5494.354,E2 -5494.354} C_VEL
LIN {X 0,Y 509.292,Z 320.105,A -85,B 0,C 180,E1 -5495.543,E2 -5495.543} C_VEL
LIN {X 0,Y 509.402,Z 314.452,A -85,B 0,C 180,E1 -5496.844,E2 -5496.844} C_VEL
LIN {X 0,Y 509.55,Z 307.322,A -85,B 0,C 180,E1 -5498.127,E2 -5498.127} C_VEL
LIN {X 0,Y 509.772,Z 299.04,A -85,B 0,C 180,E1 -5499.322,E2 -5499.322} C_VEL
LIN {X 0,Y 510.015,Z 290.552,A -85,B 0,C 180,E1 -5500.319,E2 -5500.319} C_VEL
LIN {X 0,Y 510.348,Z 280.065,A -85,B 0,C 180,E1 -5501.317,E2 -5501.317} C_VEL
LIN {X 0,Y 510.657,Z 269.087,A -85,B 0,C 180,E1 -5502.158,E2 -5502.158} C_VEL
LIN {X 0,Y 510.992,Z 258.319,A -85,B 0,C 180,E1 -5502.813,E2 -5502.813} C_VEL
LIN {X 0,Y 511.325,Z 246.66,A -85,B 0,C 180,E1 -5503.36,E2 -5503.36} C_VEL
LIN {X 0,Y 511.309,Z 235.964,A -85,B 0,C 180,E1 -5503.74,E2 -5503.74} C_VEL
LIN {X 0,Y 509.357,Z 223.36,A -85,B 0,C 180,E1 -5504.1,E2 -5504.1} C_VEL
LIN {X 0,Y 509.47,Z 214.833,A -85,B 0,C 180,E1 -5507.252,E2 -5507.252} C_VEL
LIN {X 0,Y 509.594,Z 206.71,A -85,B 0,C 180,E1 -5510.312,E2 -5510.312} C_VEL
LIN {X 0,Y 509.79,Z 198.171,A -85,B 0,C 180,E1 -5513.564,E2 -5513.564} C_VEL
LIN {X 0,Y 509.962,Z 190.945,A -85,B 0,C 180,E1 -5516.389,E2 -5516.389} C_VEL
LIN {X 0,Y 510.165,Z 183.775,A -85,B 0,C 180,E1 -5519.276,E2 -5519.276} C_VEL
LIN {X 0,Y 510.341,Z 177.187,A -85,B 0,C 180,E1 -5522.016,E2 -5522.016} C_VEL
LIN {X 0,Y 510.56,Z 170.658,A -85,B 0,C 180,E1 -5524.836,E2 -5524.836} C_VEL
LIN {X 0,Y 510.389,Z 167.421,A -85,B 0,C 180,E1 -5526.304,E2 -5526.304} C_VEL
LIN {X 0,Y 509.844,Z 163.983,A -85,B 0,C 180,E1 -5528.023,E2 -5528.023} C_VEL
LIN {X 0,Y 509.829,Z 163.979,A -85,B 0,C 180,E1 -5530.696,E2 -5530.696} C_VEL
LIN {X 0,Y 509.828,Z 163.978,A -85,B 0,C 180,E1 -5533.063,E2 -5533.063} C_VEL
LIN {X 0,Y 509.816,Z 163.98,A -85,B 0,C 180,E1 -5535.791,E2 -5535.791} C_VEL
LIN {X 0,Y 509.838,Z 163.979,A -85,B 0,C 180,E1 -5538.573,E2 -5538.573} C_VEL
LIN {X 0,Y 509.832,Z 163.981,A -85,B 0,C 180,E1 -5541.785,E2 -5541.785} C_VEL
LIN {X 0,Y 509.827,Z 163.976,A -85,B 0,C 180,E1 -5544.622,E2 -5544.622} C_VEL
LIN {X 0,Y 509.845,Z 163.976,A -85,B 0,C 180,E1 -5547.48,E2 -5547.48} C_VEL
LIN {X 0,Y 509.838,Z 163.979,A -85,B 0,C 180,E1 -5550.272,E2 -5550.272} C_VEL
LIN {X 0,Y 509.86,Z 163.974,A -85,B 0,C 180,E1 -5552.943,E2 -5552.943} C_VEL
LIN {X 0,Y 509.868,Z 163.975,A -85,B 0,C 180,E1 -5555.574,E2 -5555.574} C_VEL
LIN {X 0,Y 509.829,Z 163.976,A -85,B 0,C 180,E1 -5558.149,E2 -5558.149} C_VEL
LIN {X 0,Y 509.841,Z 163.98,A -85,B 0,C 180,E1 -5560.681,E2 -5560.681} C_VEL
LIN {X 0,Y 509.874,Z 163.972,A -85,B 0,C 180,E1 -5563.174,E2 -5563.174} C_VEL
LIN {X 0,Y 509.833,Z 163.979,A -85,B 0,C 180,E1 -5565.633,E2 -5565.633} C_VEL
LIN {X 0,Y 509.914,Z 163.971,A -85,B 0,C 180,E1 -5568.875,E2 -5568.875} C_VEL
LIN {X 0,Y 509.943,Z 163.965,A -85,B 0,C 180,E1 -5572.078,E2 -5572.078} C_VEL
LIN {X 0,Y 509.996,Z 163.958,A -85,B 0,C 180,E1 -5574.465,E2 -5574.465} C_VEL
LIN {X 0,Y 510.022,Z 163.956,A -85,B 0,C 180,E1 -5577.631,E2 -5577.631} C_VEL
LIN {X 0,Y 510.038,Z 163.954,A -85,B 0,C 180,E1 -5580.79,E2 -5580.79} C_VEL
LIN {X 0,Y 509.962,Z 163.959,A -85,B 0,C 180,E1 -5583.16,E2 -5583.16} C_VEL
LIN {X 0,Y 509.956,Z 163.962,A -85,B 0,C 180,E1 -5586.33,E2 -5586.33} C_VEL
LIN {X 0,Y 509.891,Z 163.972,A -85,B 0,C 180,E1 -5588.721,E2 -5588.721} C_VEL
LIN {X 0,Y 509.876,Z 163.973,A -85,B 0,C 180,E1 -5591.933,E2 -5591.933} C_VEL
LIN {X 0,Y 509.866,Z 163.972,A -85,B 0,C 180,E1 -5595.243,E2 -5595.243} C_VEL
LIN {X 0,Y 509.885,Z 163.971,A -85,B 0,C 180,E1 -5598.01,E2 -5598.01} C_VEL
LIN {X 0,Y 509.829,Z 163.981,A -85,B 0,C 180,E1 -5601.003,E2 -5601.003} C_VEL
LIN {X 0,Y 509.816,Z 163.98,A -85,B 0,C 180,E1 -5603.564,E2 -5603.564} C_VEL
LIN {X 0,Y 509.89,Z 163.971,A -85,B 0,C 180,E1 -5606.381,E2 -5606.381} C_VEL
LIN {X 0,Y 509.864,Z 163.973,A -85,B 0,C 180,E1 -5608.845,E2 -5608.845} C_VEL
LIN {X 0,Y 509.806,Z 163.98,A -85,B 0,C 180,E1 -5611.592,E2 -5611.592} C_VEL
LIN {X 0,Y 509.833,Z 163.98,A -85,B 0,C 180,E1 -5614.415,E2 -5614.415} C_VEL
LIN {X 0,Y 509.8,Z 163.984,A -85,B 0,C 180,E1 -5617.343,E2 -5617.343} C_VEL
LIN {X 0,Y 509.824,Z 163.978,A -85,B 0,C 180,E1 -5620.384,E2 -5620.384} C_VEL
LIN {X 0,Y 509.811,Z 163.981,A -85,B 0,C 180,E1 -5623.064,E2 -5623.064} C_VEL
LIN {X 0,Y 509.819,Z 163.98,A -85,B 0,C 180,E1 -5625.794,E2 -5625.794} C_VEL
LIN {X 0,Y 509.846,Z 163.976,A -85,B 0,C 180,E1 -5628.577,E2 -5628.577} C_VEL
LIN {X 0,Y 509.788,Z 163.984,A -85,B 0,C 180,E1 -5631.796,E2 -5631.796} C_VEL
LIN {X 0,Y 509.708,Z 164.057,A -85,B 0,C 180,E1 -5632.652,E2 -5632.652} C_VEL
LIN {X 0,Y 509.725,Z 165.651,A -85,B 0,C 180,E1 -5633.75,E2 -5633.75} C_VEL
LIN {X 0,Y 509.057,Z 166.693,A -85,B 0,C 180,E1 -5634.4,E2 -5634.4} C_VEL
LIN {X 0,Y 506.204,Z 168.582,A -85,B 0,C 180,E1 -5635.45,E2 -5635.45} C_VEL
LIN {X 0,Y 503.781,Z 170.119,A -85,B 0,C 180,E1 -5636.296,E2 -5636.296} C_VEL
LIN {X 0,Y 502.723,Z 171.212,A -85,B 0,C 180,E1 -5636.95,E2 -5636.95} C_VEL
LIN {X 0,Y 502.627,Z 171.554,A -85,B 0,C 180,E1 -5637.173,E2 -5637.173} C_VEL
LIN {X 0,Y 502.53,Z 175.999,A -85,B 0,C 180,E1 -5640.122,E2 -5640.122} C_VEL
LIN {X 0,Y 502.434,Z 179.669,A -85,B 0,C 180,E1 -5642.511,E2 -5642.511} C_VEL
LIN {X 0,Y 502.399,Z 184.186,A -85,B 0,C 180,E1 -5645.407,E2 -5645.407} C_VEL
LIN {X 0,Y 502.289,Z 188.011,A -85,B 0,C 180,E1 -5647.805,E2 -5647.805} C_VEL
LIN {X 0,Y 502.249,Z 192.247,A -85,B 0,C 180,E1 -5650.378,E2 -5650.378} C_VEL
LIN {X 0,Y 502.179,Z 196.453,A -85,B 0,C 180,E1 -5652.909,E2 -5652.909} C_VEL
LIN {X 0,Y 502.185,Z 197.891,A -85,B 0,C 180,E1 -5653.765,E2 -5653.765} C_VEL
LIN {X 0,Y 504.676,Z 211.346,A -85,B 0,C 180,E1 -5654.214,E2 -5654.214} C_VEL
LIN {X 0,Y 504.388,Z 223.694,A -85,B 0,C 180,E1 -5654.701,E2 -5654.701} C_VEL
LIN {X 0,Y 504.042,Z 236.006,A -85,B 0,C 180,E1 -5655.362,E2 -5655.362} C_VEL
LIN {X 0,Y 503.628,Z 247.599,A -85,B 0,C 180,E1 -5656.174,E2 -5656.174} C_VEL
LIN {X 0,Y 503.338,Z 258.016,A -85,B 0,C 180,E1 -5657.091,E2 -5657.091} C_VEL
LIN {X 0,Y 502.984,Z 267.64,A -85,B 0,C 180,E1 -5658.142,E2 -5658.142} C_VEL
LIN {X 0,Y 502.767,Z 276.376,A -85,B 0,C 180,E1 -5659.326,E2 -5659.326} C_VEL
LIN {X 0,Y 502.508,Z 283.627,A -85,B 0,C 180,E1 -5660.542,E2 -5660.542} C_VEL
LIN {X 0,Y 502.348,Z 288.519,A -85,B 0,C 180,E1 -5661.553,E2 -5661.553} C_VEL
LIN {X 0,Y 502.246,Z 293.264,A -85,B 0,C 180,E1 -5662.765,E2 -5662.765} C_VEL
LIN {X 0,Y 502.156,Z 296.458,A -85,B 0,C 180,E1 -5663.808,E2 -5663.808} C_VEL
LIN {X 0,Y 502.067,Z 299.514,A -85,B 0,C 180,E1 -5665.182,E2 -5665.182} C_VEL
LIN {X 0,Y 502.128,Z 300.744,A -85,B 0,C 180,E1 -5665.987,E2 -5665.987} C_VEL
LIN {X 0,Y 502.112,Z 301.57,A -85,B 0,C 180,E1 -5666.79,E2 -5666.79} C_VEL
LIN {X 0,Y 502.091,Z 301.97,A -85,B 0,C 180,E1 -5667.593,E2 -5667.593} C_VEL
LIN {X 0,Y 501.992,Z 301.633,A -85,B 0,C 180,E1 -5669.197,E2 -5669.197} C_VEL
LIN {X 0,Y 501.987,Z 300.885,A -85,B 0,C 180,E1 -5669.999,E2 -5669.999} C_VEL
LIN {X 0,Y 502.068,Z 298.118,A -85,B 0,C 180,E1 -5671.604,E2 -5671.604} C_VEL
LIN {X 0,Y 502.216,Z 294.94,A -85,B 0,C 180,E1 -5672.807,E2 -5672.807} C_VEL
LIN {X 0,Y 502.305,Z 290.716,A -85,B 0,C 180,E1 -5674.011,E2 -5674.011} C_VEL
LIN {X 0,Y 502.528,Z 285.318,A -85,B 0,C 180,E1 -5675.215,E2 -5675.215} C_VEL
LIN {X 0,Y 502.682,Z 278.583,A -85,B 0,C 180,E1 -5676.421,E2 -5676.421} C_VEL
LIN {X 0,Y 502.894,Z 270.2,A -85,B 0,C 180,E1 -5677.628,E2 -5677.628} C_VEL
LIN {X 0,Y 503.284,Z 261.567,A -85,B 0,C 180,E1 -5678.632,E2 -5678.632} C_VEL
LIN {X 0,Y 503.631,Z 250.953,A -85,B 0,C 180,E1 -5679.639,E2 -5679.639} C_VEL
LIN {X 0,Y 503.915,Z 240.389,A -85,B 0,C 180,E1 -5680.445,E2 -5680.445} C_VEL
LIN {X 0,Y 504.255,Z 228.568,A -85,B 0,C 180,E1 -5681.149,E2 -5681.149} C_VEL
LIN {X 0,Y 504.599,Z 215.511,A -85,B 0,C 180,E1 -5681.731,E2 -5681.731} C_VEL
LIN {X 0,Y 504.47,Z 209.425,A -85,B 0,C 180,E1 -5681.947,E2 -5681.947} C_VEL
LIN {X 0,Y 502.187,Z 197.88,A -85,B 0,C 180,E1 -5682.324,E2 -5682.324} C_VEL
LIN {X 0,Y 502.283,Z 192.704,A -85,B 0,C 180,E1 -5685.416,E2 -5685.416} C_VEL
LIN {X 0,Y 502.317,Z 188.528,A -85,B 0,C 180,E1 -5687.935,E2 -5687.935} C_VEL
LIN {X 0,Y 502.412,Z 184.451,A -85,B 0,C 180,E1 -5690.468,E2 -5690.468} C_VEL
LIN {X 0,Y 502.412,Z 180.362,A -85,B 0,C 180,E1 -5693.057,E2 -5693.057} C_VEL
LIN {X 0,Y 502.471,Z 176.261,A -85,B 0,C 180,E1 -5695.693,E2 -5695.693} C_VEL
LIN {X 0,Y 502.564,Z 172.136,A -85,B 0,C 180,E1 -5698.387,E2 -5698.387} C_VEL
LIN {X 0,Y 502.68,Z 167.985,A -85,B 0,C 180,E1 -5701.148,E2 -5701.148} C_VEL
LIN {X 0,Y 502.645,Z 165.203,A -85,B 0,C 180,E1 -5703.042,E2 -5703.042} C_VEL
LIN {X 0,Y 502.775,Z 164.86,A -85,B 0,C 180,E1 -5704.964,E2 -5704.964} C_VEL
LIN {X 0,Y 502.78,Z 164.858,A -85,B 0,C 180,E1 -5708.483,E2 -5708.483} C_VEL
LIN {X 0,Y 502.806,Z 164.852,A -85,B 0,C 180,E1 -5711.063,E2 -5711.063} C_VEL
LIN {X 0,Y 502.765,Z 164.86,A -85,B 0,C 180,E1 -5713.373,E2 -5713.373} C_VEL
LIN {X 0,Y 502.771,Z 164.858,A -85,B 0,C 180,E1 -5715.658,E2 -5715.658} C_VEL
LIN {X 0,Y 502.819,Z 164.849,A -85,B 0,C 180,E1 -5717.862,E2 -5717.862} C_VEL
LIN {X 0,Y 502.786,Z 164.857,A -85,B 0,C 180,E1 -5721.022,E2 -5721.022} C_VEL
LIN {X 0,Y 502.752,Z 164.862,A -85,B 0,C 180,E1 -5724.166,E2 -5724.166} C_VEL
LIN {X 0,Y 502.806,Z 164.853,A -85,B 0,C 180,E1 -5726.991,E2 -5726.991} C_VEL
LIN {X 0,Y 502.802,Z 164.853,A -85,B 0,C 180,E1 -5730.059,E2 -5730.059} C_VEL
LIN {X 0,Y 502.809,Z 164.853,A -85,B 0,C 180,E1 -5732.531,E2 -5732.531} C_VEL
LIN {X 0,Y 502.813,Z 164.85,A -85,B 0,C 180,E1 -5735.292,E2 -5735.292} C_VEL
LIN {X 0,Y 502.788,Z 164.855,A -85,B 0,C 180,E1 -5737.826,E2 -5737.826} C_VEL
LIN {X 0,Y 502.789,Z 164.855,A -85,B 0,C 180,E1 -5740.398,E2 -5740.398} C_VEL
LIN {X 0,Y 502.805,Z 164.854,A -85,B 0,C 180,E1 -5742.93,E2 -5742.93} C_VEL
LIN {X 0,Y 502.822,Z 164.853,A -85,B 0,C 180,E1 -5745.428,E2 -5745.428} C_VEL
LIN {X 0,Y 502.89,Z 164.844,A -85,B 0,C 180,E1 -5748.717,E2 -5748.717} C_VEL
LIN {X 0,Y 502.907,Z 164.843,A -85,B 0,C 180,E1 -5751.967,E2 -5751.967} C_VEL
LIN {X 0,Y 502.94,Z 164.835,A -85,B 0,C 180,E1 -5754.386,E2 -5754.386} C_VEL
LIN {X 0,Y 502.985,Z 164.833,A -85,B 0,C 180,E1 -5757.597,E2 -5757.597} C_VEL
LIN {X 0,Y 502.982,Z 164.83,A -85,B 0,C 180,E1 -5760,E2 -5760} C_VEL
LIN {X 0,Y 502.992,Z 164.832,A -85,B 0,C 180,E1 -5762.402,E2 -5762.402} C_VEL
LIN {X 0,Y 502.939,Z 164.837,A -85,B 0,C 180,E1 -5765.613,E2 -5765.613} C_VEL
LIN {X 0,Y 502.907,Z 164.841,A -85,B 0,C 180,E1 -5768.033,E2 -5768.033} C_VEL
LIN {X 0,Y 502.875,Z 164.849,A -85,B 0,C 180,E1 -5771.283,E2 -5771.283} C_VEL
LIN {X 0,Y 502.816,Z 164.853,A -85,B 0,C 180,E1 -5774.572,E2 -5774.572} C_VEL
LIN {X 0,Y 502.825,Z 164.853,A -85,B 0,C 180,E1 -5777.908,E2 -5777.908} C_VEL
LIN {X 0,Y 502.796,Z 164.854,A -85,B 0,C 180,E1 -5780.538,E2 -5780.538} C_VEL
LIN {X 0,Y 502.789,Z 164.856,A -85,B 0,C 180,E1 -5783.041,E2 -5783.041} C_VEL
LIN {X 0,Y 502.823,Z 164.85,A -85,B 0,C 180,E1 -5785.676,E2 -5785.676} C_VEL
LIN {X 0,Y 502.813,Z 164.852,A -85,B 0,C 180,E1 -5788.374,E2 -5788.374} C_VEL
LIN {X 0,Y 502.767,Z 164.857,A -85,B 0,C 180,E1 -5791.502,E2 -5791.502} C_VEL
LIN {X 0,Y 502.776,Z 164.857,A -85,B 0,C 180,E1 -5794.446,E2 -5794.446} C_VEL
LIN {X 0,Y 502.754,Z 164.862,A -85,B 0,C 180,E1 -5797.181,E2 -5797.181} C_VEL
LIN {X 0,Y 502.803,Z 164.852,A -85,B 0,C 180,E1 -5800.014,E2 -5800.014} C_VEL
LIN {X 0,Y 502.804,Z 164.853,A -85,B 0,C 180,E1 -5802.205,E2 -5802.205} C_VEL
LIN {X 0,Y 502.78,Z 164.854,A -85,B 0,C 180,E1 -5805.471,E2 -5805.471} C_VEL
LIN {X 0,Y 502.815,Z 164.857,A -85,B 0,C 180,E1 -5807.867,E2 -5807.867} C_VEL
LIN {X 0,Y 502.784,Z 164.86,A -85,B 0,C 180,E1 -5811.026,E2 -5811.026} C_VEL
LIN {X 0,Y 502.785,Z 164.925,A -85,B 0,C 180,E1 -5812.149,E2 -5812.149} C_VEL
LIN {X 0,Y 503.538,Z 170.193,A -85,B 0,C 180,E1 -5814.608,E2 -5814.608} C_VEL
LIN {X 0,Y 503.305,Z 176.814,A -85,B 0,C 180,E1 -5817.483,E2 -5817.483} C_VEL
LIN {X 0,Y 503.142,Z 184.58,A -85,B 0,C 180,E1 -5820.735,E2 -5820.735} C_VEL
LIN {X 0,Y 502.856,Z 193.52,A -85,B 0,C 180,E1 -5824.328,E2 -5824.328} C_VEL
LIN {X 0,Y 502.658,Z 201.216,A -85,B 0,C 180,E1 -5827.338,E2 -5827.338} C_VEL
LIN {X 0,Y 502.49,Z 209.161,A -85,B 0,C 180,E1 -5830.389,E2 -5830.389} C_VEL
LIN {X 0,Y 502.372,Z 216.947,A -85,B 0,C 180,E1 -5833.336,E2 -5833.336} C_VEL
LIN {X 0,Y 502.299,Z 223.229,A -85,B 0,C 180,E1 -5835.699,E2 -5835.699} C_VEL
LIN {X 0,Y 504.465,Z 237.417,A -85,B 0,C 180,E1 -5836.122,E2 -5836.122} C_VEL
LIN {X 0,Y 504.301,Z 249.975,A -85,B 0,C 180,E1 -5836.605,E2 -5836.605} C_VEL
LIN {X 0,Y 503.956,Z 261.517,A -85,B 0,C 180,E1 -5837.201,E2 -5837.201} C_VEL
LIN {X 0,Y 503.603,Z 272.365,A -85,B 0,C 180,E1 -5837.918,E2 -5837.918} C_VEL
LIN {X 0,Y 503.278,Z 283.274,A -85,B 0,C 180,E1 -5838.829,E2 -5838.829} C_VEL
LIN {X 0,Y 502.935,Z 292.169,A -85,B 0,C 180,E1 -5839.738,E2 -5839.738} C_VEL
LIN {X 0,Y 502.65,Z 301.837,A -85,B 0,C 180,E1 -5840.951,E2 -5840.951} C_VEL
LIN {X 0,Y 502.4,Z 309.532,A -85,B 0,C 180,E1 -5842.162,E2 -5842.162} C_VEL
LIN {X 0,Y 502.234,Z 316.627,A -85,B 0,C 180,E1 -5843.573,E2 -5843.573} C_VEL
LIN {X 0,Y 502.179,Z 321.348,A -85,B 0,C 180,E1 -5844.782,E2 -5844.782} C_VEL
LIN {X 0,Y 502.138,Z 324.954,A -85,B 0,C 180,E1 -5845.988,E2 -5845.988} C_VEL
LIN {X 0,Y 502.12,Z 326.814,A -85,B 0,C 180,E1 -5846.791,E2 -5846.791} C_VEL
LIN {X 0,Y 502.091,Z 328.208,A -85,B 0,C 180,E1 -5847.594,E2 -5847.594} C_VEL
LIN {X 0,Y 501.991,Z 329.808,A -85,B 0,C 180,E1 -5849.198,E2 -5849.198} C_VEL
LIN {X 0,Y 501.982,Z 330.024,A -85,B 0,C 180,E1 -5850.001,E2 -5850.001} C_VEL
LIN {X 0,Y 502.036,Z 329.201,A -85,B 0,C 180,E1 -5851.605,E2 -5851.605} C_VEL
LIN {X 0,Y 502.092,Z 328.208,A -85,B 0,C 180,E1 -5852.407,E2 -5852.407} C_VEL
LIN {X 0,Y 502.12,Z 326.813,A -85,B 0,C 180,E1 -5853.21,E2 -5853.21} C_VEL
LIN {X 0,Y 502.102,Z 323.877,A -85,B 0,C 180,E1 -5854.415,E2 -5854.415} C_VEL
LIN {X 0,Y 502.208,Z 319.907,A -85,B 0,C 180,E1 -5855.622,E2 -5855.622} C_VEL
LIN {X 0,Y 502.332,Z 313.9,A -85,B 0,C 180,E1 -5857.012,E2 -5857.012} C_VEL
LIN {X 0,Y 502.481,Z 307.122,A -85,B 0,C 180,E1 -5858.242,E2 -5858.242} C_VEL
LIN {X 0,Y 502.734,Z 298.84,A -85,B 0,C 180,E1 -5859.454,E2 -5859.454} C_VEL
LIN {X 0,Y 502.995,Z 290.352,A -85,B 0,C 180,E1 -5860.465,E2 -5860.465} C_VEL
LIN {X 0,Y 503.368,Z 279.866,A -85,B 0,C 180,E1 -5861.476,E2 -5861.476} C_VEL
LIN {X 0,Y 503.675,Z 268.887,A -85,B 0,C 180,E1 -5862.329,E2 -5862.329} C_VEL
LIN {X 0,Y 504.037,Z 258.12,A -85,B 0,C 180,E1 -5862.993,E2 -5862.993} C_VEL
LIN {X 0,Y 504.408,Z 246.461,A -85,B 0,C 180,E1 -5863.547,E2 -5863.547} C_VEL
LIN {X 0,Y 504.407,Z 236.983,A -85,B 0,C 180,E1 -5863.894,E2 -5863.894} C_VEL
LIN {X 0,Y 502.398,Z 224.229,A -85,B 0,C 180,E1 -5864.273,E2 -5864.273} C_VEL
LIN {X 0,Y 502.294,Z 223.129,A -85,B 0,C 180,E1 -5864.328,E2 -5864.328} C_VEL
LIN {X 0,Y 502.399,Z 214.69,A -85,B 0,C 180,E1 -5867.503,E2 -5867.503} C_VEL
LIN {X 0,Y 502.544,Z 206.971,A -85,B 0,C 180,E1 -5870.463,E2 -5870.463} C_VEL
LIN {X 0,Y 502.716,Z 199.176,A -85,B 0,C 180,E1 -5873.479,E2 -5873.479} C_VEL
LIN {X 0,Y 502.914,Z 191.388,A -85,B 0,C 180,E1 -5876.572,E2 -5876.572} C_VEL
LIN {X 0,Y 503.137,Z 184.806,A -85,B 0,C 180,E1 -5879.266,E2 -5879.266} C_VEL
LIN {X 0,Y 503.333,Z 178.239,A -85,B 0,C 180,E1 -5882.043,E2 -5882.043} C_VEL
LIN {X 0,Y 503.555,Z 171.707,A -85,B 0,C 180,E1 -5884.903,E2 -5884.903} C_VEL
LIN {X 0,Y 503.241,Z 167.403,A -85,B 0,C 180,E1 -5886.904,E2 -5886.904} C_VEL
LIN {X 0,Y 502.808,Z 164.859,A -85,B 0,C 180,E1 -5888.216,E2 -5888.216} C_VEL
LIN {X 0,Y 502.809,Z 164.852,A -85,B 0,C 180,E1 -5891.064,E2 -5891.064} C_VEL
LIN {X 0,Y 502.77,Z 164.859,A -85,B 0,C 180,E1 -5893.374,E2 -5893.374} C_VEL
LIN {X 0,Y 502.775,Z 164.858,A -85,B 0,C 180,E1 -5895.659,E2 -5895.659} C_VEL
LIN {X 0,Y 502.801,Z 164.855,A -85,B 0,C 180,E1 -5899.003,E2 -5899.003} C_VEL
LIN {X 0,Y 502.775,Z 164.859,A -85,B 0,C 180,E1 -5902.044,E2 -5902.044} C_VEL
LIN {X 0,Y 502.791,Z 164.855,A -85,B 0,C 180,E1 -5905.033,E2 -5905.033} C_VEL
LIN {X 0,Y 502.767,Z 164.857,A -85,B 0,C 180,E1 -5907.914,E2 -5907.914} C_VEL
LIN {X 0,Y 502.804,Z 164.856,A -85,B 0,C 180,E1 -5910.711,E2 -5910.711} C_VEL
LIN {X 0,Y 502.839,Z 164.851,A -85,B 0,C 180,E1 -5913.438,E2 -5913.438} C_VEL
LIN {X 0,Y 502.793,Z 164.853,A -85,B 0,C 180,E1 -5916.086,E2 -5916.086} C_VEL
LIN {X 0,Y 502.776,Z 164.859,A -85,B 0,C 180,E1 -5918.689,E2 -5918.689} C_VEL
LIN {X 0,Y 502.837,Z 164.85,A -85,B 0,C 180,E1 -5921.87,E2 -5921.87} C_VEL
LIN {X 0,Y 502.812,Z 164.852,A -85,B 0,C 180,E1 -5924.661,E2 -5924.661} C_VEL
LIN {X 0,Y 502.874,Z 164.844,A -85,B 0,C 180,E1 -5928.024,E2 -5928.024} C_VEL
LIN {X 0,Y 502.874,Z 164.843,A -85,B 0,C 180,E1 -5931.157,E2 -5931.157} C_VEL
LIN {X 0,Y 502.934,Z 164.837,A -85,B 0,C 180,E1 -5933.582,E2 -5933.582} C_VEL
LIN {X 0,Y 502.874,Z 164.845,A -85,B 0,C 180,E1 -5936.796,E2 -5936.796} C_VEL
LIN {X 0,Y 503.003,Z 164.83,A -85,B 0,C 180,E1 -5939.2,E2 -5939.2} C_VEL
LIN {X 0,Y 502.873,Z 164.843,A -85,B 0,C 180,E1 -5941.602,E2 -5941.602} C_VEL
LIN {X 0,Y 502.904,Z 164.838,A -85,B 0,C 180,E1 -5943.205,E2 -5943.205} C_VEL
LIN {X 0,Y 502.905,Z 164.84,A -85,B 0,C 180,E1 -5946.419,E2 -5946.419} C_VEL
LIN {X 0,Y 502.849,Z 164.849,A -85,B 0,C 180,E1 -5948.844,E2 -5948.844} C_VEL
LIN {X 0,Y 502.818,Z 164.854,A -85,B 0,C 180,E1 -5952.103,E2 -5952.103} C_VEL
LIN {X 0,Y 502.822,Z 164.851,A -85,B 0,C 180,E1 -5955.401,E2 -5955.401} C_VEL
LIN {X 0,Y 502.838,Z 164.848,A -85,B 0,C 180,E1 -5958.13,E2 -5958.13} C_VEL
LIN {X 0,Y 502.768,Z 164.859,A -85,B 0,C 180,E1 -5961.312,E2 -5961.312} C_VEL
LIN {X 0,Y 502.77,Z 164.86,A -85,B 0,C 180,E1 -5963.915,E2 -5963.915} C_VEL
LIN {X 0,Y 502.842,Z 164.848,A -85,B 0,C 180,E1 -5966.568,E2 -5966.568} C_VEL
LIN {X 0,Y 502.818,Z 164.856,A -85,B 0,C 180,E1 -5969.289,E2 -5969.289} C_VEL
LIN {X 0,Y 502.768,Z 164.857,A -85,B 0,C 180,E1 -5972.086,E2 -5972.086} C_VEL
LIN {X 0,Y 502.789,Z 164.855,A -85,B 0,C 180,E1 -5974.967,E2 -5974.967} C_VEL
LIN {X 0,Y 502.776,Z 164.858,A -85,B 0,C 180,E1 -5977.956,E2 -5977.956} C_VEL
LIN {X 0,Y 502.806,Z 164.856,A -85,B 0,C 180,E1 -5981.068,E2 -5981.068} C_VEL
LIN {X 0,Y 502.789,Z 164.859,A -85,B 0,C 180,E1 -5984.534,E2 -5984.534} C_VEL
LIN {X 0,Y 502.785,Z 164.857,A -85,B 0,C 180,E1 -5987.863,E2 -5987.863} C_VEL
LIN {X 0,Y 502.769,Z 164.857,A -85,B 0,C 180,E1 -5990.249,E2 -5990.249} C_VEL
LIN {X 0,Y 502.725,Z 164.864,A -85,B 0,C 180,E1 -5992.043,E2 -5992.043} C_VEL
LIN {X 0,Y 502.664,Z 165.539,A -85,B 0,C 180,E1 -5993.046,E2 -5993.046} C_VEL
LIN {X 0,Y 502.651,Z 169.819,A -85,B 0,C 180,E1 -5995.996,E2 -5995.996} C_VEL
LIN {X 0,Y 502.627,Z 171.554,A -85,B 0,C 180,E1 -5997.173,E2 -5997.173} C_VEL
LIN {X 0,Y 501.931,Z 172.619,A -85,B 0,C 180,E1 -5997.83,E2 -5997.83} C_VEL
LIN {X 0,Y 499.043,Z 174.539,A -85,B 0,C 180,E1 -5998.894,E2 -5998.894} C_VEL
LIN {X 0,Y 496.606,Z 176.095,A -85,B 0,C 180,E1 -5999.75,E2 -5999.75} C_VEL
LIN {X 0,Y 495.546,Z 177.209,A -85,B 0,C 180,E1 -6000.413,E2 -6000.413} C_VEL
LIN {X 0,Y 495.453,Z 177.557,A -85,B 0,C 180,E1 -6000.639,E2 -6000.639} C_VEL
LIN {X 0,Y 495.356,Z 181.703,A -85,B 0,C 180,E1 -6003.36,E2 -6003.36} C_VEL
LIN {X 0,Y 495.306,Z 185.333,A -85,B 0,C 180,E1 -6005.703,E2 -6005.703} C_VEL
LIN {X 0,Y 495.193,Z 189.536,A -85,B 0,C 180,E1 -6008.347,E2 -6008.347} C_VEL
LIN {X 0,Y 495.159,Z 193.776,A -85,B 0,C 180,E1 -6010.948,E2 -6010.948} C_VEL
LIN {X 0,Y 495.119,Z 198.224,A -85,B 0,C 180,E1 -6013.57,E2 -6013.57} C_VEL
LIN {X 0,Y 497.683,Z 211.397,A -85,B 0,C 180,E1 -6014.008,E2 -6014.008} C_VEL
LIN {X 0,Y 497.477,Z 224.445,A -85,B 0,C 180,E1 -6014.535,E2 -6014.535} C_VEL
LIN {X 0,Y 497.165,Z 235.79,A -85,B 0,C 180,E1 -6015.155,E2 -6015.155} C_VEL
LIN {X 0,Y 496.675,Z 247.454,A -85,B 0,C 180,E1 -6015.977,E2 -6015.977} C_VEL
LIN {X 0,Y 496.387,Z 257.925,A -85,B 0,C 180,E1 -6016.907,E2 -6016.907} C_VEL
LIN {X 0,Y 496.035,Z 266.67,A -85,B 0,C 180,E1 -6017.857,E2 -6017.857} C_VEL
LIN {X 0,Y 495.789,Z 275.035,A -85,B 0,C 180,E1 -6018.968,E2 -6018.968} C_VEL
LIN {X 0,Y 495.441,Z 282.557,A -85,B 0,C 180,E1 -6020.199,E2 -6020.199} C_VEL
LIN {X 0,Y 495.31,Z 288.593,A -85,B 0,C 180,E1 -6021.432,E2 -6021.432} C_VEL
LIN {X 0,Y 495.171,Z 293.364,A -85,B 0,C 180,E1 -6022.661,E2 -6022.661} C_VEL
LIN {X 0,Y 495.128,Z 296.056,A -85,B 0,C 180,E1 -6023.52,E2 -6023.52} C_VEL
LIN {X 0,Y 495.076,Z 298.017,A -85,B 0,C 180,E1 -6024.297,E2 -6024.297} C_VEL
LIN {X 0,Y 495.025,Z 300.904,A -85,B 0,C 180,E1 -6025.929,E2 -6025.929} C_VEL
LIN {X 0,Y 495.034,Z 301.748,A -85,B 0,C 180,E1 -6026.744,E2 -6026.744} C_VEL
LIN {X 0,Y 494.963,Z 302.194,A -85,B 0,C 180,E1 -6028.372,E2 -6028.372} C_VEL
LIN {X 0,Y 494.905,Z 301.115,A -85,B 0,C 180,E1 -6029.999,E2 -6029.999} C_VEL
LIN {X 0,Y 494.92,Z 299.948,A -85,B 0,C 180,E1 -6030.813,E2 -6030.813} C_VEL
LIN {X 0,Y 494.993,Z 298.376,A -85,B 0,C 180,E1 -6031.627,E2 -6031.627} C_VEL
LIN {X 0,Y 495.153,Z 295.222,A -85,B 0,C 180,E1 -6032.847,E2 -6032.847} C_VEL
LIN {X 0,Y 495.248,Z 291.023,A -85,B 0,C 180,E1 -6034.068,E2 -6034.068} C_VEL
LIN {X 0,Y 495.434,Z 284.658,A -85,B 0,C 180,E1 -6035.494,E2 -6035.494} C_VEL
LIN {X 0,Y 495.657,Z 278.948,A -85,B 0,C 180,E1 -6036.512,E2 -6036.512} C_VEL
LIN {X 0,Y 495.87,Z 270.618,A -85,B 0,C 180,E1 -6037.737,E2 -6037.737} C_VEL
LIN {X 0,Y 496.298,Z 262.027,A -85,B 0,C 180,E1 -6038.755,E2 -6038.755} C_VEL
LIN {X 0,Y 496.668,Z 251.463,A -85,B 0,C 180,E1 -6039.775,E2 -6039.775} C_VEL
LIN {X 0,Y 496.954,Z 240.965,A -85,B 0,C 180,E1 -6040.593,E2 -6040.593} C_VEL
LIN {X 0,Y 497.329,Z 229.277,A -85,B 0,C 180,E1 -6041.306,E2 -6041.306} C_VEL
LIN {X 0,Y 497.695,Z 216.729,A -85,B 0,C 180,E1 -6041.881,E2 -6041.881} C_VEL
LIN {X 0,Y 497.596,Z 210.384,A -85,B 0,C 180,E1 -6042.114,E2 -6042.114} C_VEL
LIN {X 0,Y 495.128,Z 198.066,A -85,B 0,C 180,E1 -6042.526,E2 -6042.526} C_VEL
LIN {X 0,Y 495.197,Z 192.905,A -85,B 0,C 180,E1 -6045.642,E2 -6045.642} C_VEL
LIN {X 0,Y 495.237,Z 188.728,A -85,B 0,C 180,E1 -6048.19,E2 -6048.19} C_VEL
LIN {X 0,Y 495.33,Z 184.622,A -85,B 0,C 180,E1 -6050.774,E2 -6050.774} C_VEL
LIN {X 0,Y 495.339,Z 180.514,A -85,B 0,C 180,E1 -6053.405,E2 -6053.405} C_VEL
LIN {X 0,Y 495.423,Z 176.404,A -85,B 0,C 180,E1 -6056.086,E2 -6056.086} C_VEL
LIN {X 0,Y 495.525,Z 172.271,A -85,B 0,C 180,E1 -6058.828,E2 -6058.828} C_VEL
LIN {X 0,Y 495.657,Z 168.013,A -85,B 0,C 180,E1 -6061.706,E2 -6061.706} C_VEL
LIN {X 0,Y 495.601,Z 165.833,A -85,B 0,C 180,E1 -6063.209,E2 -6063.209} C_VEL
LIN {X 0,Y 495.73,Z 165.735,A -85,B 0,C 180,E1 -6065.536,E2 -6065.536} C_VEL
LIN {X 0,Y 495.748,Z 165.735,A -85,B 0,C 180,E1 -6068.765,E2 -6068.765} C_VEL
LIN {X 0,Y 495.762,Z 165.734,A -85,B 0,C 180,E1 -6071.776,E2 -6071.776} C_VEL
LIN {X 0,Y 495.731,Z 165.735,A -85,B 0,C 180,E1 -6075.137,E2 -6075.137} C_VEL
LIN {X 0,Y 495.765,Z 165.727,A -85,B 0,C 180,E1 -6078.219,E2 -6078.219} C_VEL
LIN {X 0,Y 495.745,Z 165.732,A -85,B 0,C 180,E1 -6081.228,E2 -6081.228} C_VEL
LIN {X 0,Y 495.725,Z 165.738,A -85,B 0,C 180,E1 -6084.46,E2 -6084.46} C_VEL
LIN {X 0,Y 495.742,Z 165.736,A -85,B 0,C 180,E1 -6087.403,E2 -6087.403} C_VEL
LIN {X 0,Y 495.754,Z 165.73,A -85,B 0,C 180,E1 -6090.252,E2 -6090.252} C_VEL
LIN {X 0,Y 495.804,Z 165.725,A -85,B 0,C 180,E1 -6093.246,E2 -6093.246} C_VEL
LIN {X 0,Y 495.745,Z 165.73,A -85,B 0,C 180,E1 -6095.724,E2 -6095.724} C_VEL
LIN {X 0,Y 495.733,Z 165.736,A -85,B 0,C 180,E1 -6098.37,E2 -6098.37} C_VEL
LIN {X 0,Y 495.749,Z 165.732,A -85,B 0,C 180,E1 -6100.97,E2 -6100.97} C_VEL
LIN {X 0,Y 495.749,Z 165.734,A -85,B 0,C 180,E1 -6103.529,E2 -6103.529} C_VEL
LIN {X 0,Y 495.776,Z 165.728,A -85,B 0,C 180,E1 -6106.055,E2 -6106.055} C_VEL
LIN {X 0,Y 495.863,Z 165.721,A -85,B 0,C 180,E1 -6108.555,E2 -6108.555} C_VEL
LIN {X 0,Y 495.868,Z 165.719,A -85,B 0,C 180,E1 -6111.852,E2 -6111.852} C_VEL
LIN {X 0,Y 495.895,Z 165.713,A -85,B 0,C 180,E1 -6114.306,E2 -6114.306} C_VEL
LIN {X 0,Y 495.955,Z 165.709,A -85,B 0,C 180,E1 -6117.563,E2 -6117.563} C_VEL
LIN {X 0,Y 495.954,Z 165.706,A -85,B 0,C 180,E1 -6120,E2 -6120} C_VEL
LIN {X 0,Y 495.962,Z 165.707,A -85,B 0,C 180,E1 -6122.436,E2 -6122.436} C_VEL
LIN {X 0,Y 495.893,Z 165.716,A -85,B 0,C 180,E1 -6125.693,E2 -6125.693} C_VEL
LIN {X 0,Y 495.867,Z 165.717,A -85,B 0,C 180,E1 -6128.148,E2 -6128.148} C_VEL
LIN {X 0,Y 495.845,Z 165.722,A -85,B 0,C 180,E1 -6131.445,E2 -6131.445} C_VEL
LIN {X 0,Y 495.759,Z 165.733,A -85,B 0,C 180,E1 -6134.784,E2 -6134.784} C_VEL
LIN {X 0,Y 495.751,Z 165.731,A -85,B 0,C 180,E1 -6137.32,E2 -6137.32} C_VEL
LIN {X 0,Y 495.742,Z 165.735,A -85,B 0,C 180,E1 -6139.891,E2 -6139.891} C_VEL
LIN {X 0,Y 495.757,Z 165.731,A -85,B 0,C 180,E1 -6142.871,E2 -6142.871} C_VEL
LIN {X 0,Y 495.775,Z 165.726,A -85,B 0,C 180,E1 -6146.069,E2 -6146.069} C_VEL
LIN {X 0,Y 495.752,Z 165.735,A -85,B 0,C 180,E1 -6148.816,E2 -6148.816} C_VEL
LIN {X 0,Y 495.729,Z 165.735,A -85,B 0,C 180,E1 -6151.728,E2 -6151.728} C_VEL
LIN {X 0,Y 495.746,Z 165.732,A -85,B 0,C 180,E1 -6154.697,E2 -6154.697} C_VEL
LIN {X 0,Y 495.707,Z 165.739,A -85,B 0,C 180,E1 -6157.564,E2 -6157.564} C_VEL
LIN {X 0,Y 495.77,Z 165.728,A -85,B 0,C 180,E1 -6160.054,E2 -6160.054} C_VEL
LIN {X 0,Y 495.742,Z 165.733,A -85,B 0,C 180,E1 -6162.881,E2 -6162.881} C_VEL
LIN {X 0,Y 495.717,Z 165.739,A -85,B 0,C 180,E1 -6166.002,E2 -6166.002} C_VEL
LIN {X 0,Y 495.747,Z 165.735,A -85,B 0,C 180,E1 -6168.708,E2 -6168.708} C_VEL
LIN {X 0,Y 495.782,Z 165.857,A -85,B 0,C 180,E1 -6171.997,E2 -6171.997} C_VEL
LIN {X 0,Y 496.517,Z 171.195,A -85,B 0,C 180,E1 -6174.529,E2 -6174.529} C_VEL
LIN {X 0,Y 496.371,Z 175.978,A -85,B 0,C 180,E1 -6176.654,E2 -6176.654} C_VEL
LIN {X 0,Y 496.173,Z 183.248,A -85,B 0,C 180,E1 -6179.772,E2 -6179.772} C_VEL
LIN {X 0,Y 495.876,Z 190.027,A -85,B 0,C 180,E1 -6182.576,E2 -6182.576} C_VEL
LIN {X 0,Y 495.746,Z 196.368,A -85,B 0,C 180,E1 -6185.136,E2 -6185.136} C_VEL
LIN {X 0,Y 495.554,Z 204.547,A -85,B 0,C 180,E1 -6188.365,E2 -6188.365} C_VEL
LIN {X 0,Y 495.383,Z 212.335,A -85,B 0,C 180,E1 -6191.387,E2 -6191.387} C_VEL
LIN {X 0,Y 495.242,Z 220.085,A -85,B 0,C 180,E1 -6194.36,E2 -6194.36} C_VEL
LIN {X 0,Y 495.212,Z 223.177,A -85,B 0,C 180,E1 -6195.503,E2 -6195.503} C_VEL
LIN {X 0,Y 497.251,Z 236.407,A -85,B 0,C 180,E1 -6195.89,E2 -6195.89} C_VEL
LIN {X 0,Y 497.608,Z 241.009,A -85,B 0,C 180,E1 -6196.057,E2 -6196.057} C_VEL
LIN {X 0,Y 497.228,Z 254.033,A -85,B 0,C 180,E1 -6196.619,E2 -6196.619} C_VEL
LIN {X 0,Y 496.809,Z 266.284,A -85,B 0,C 180,E1 -6197.332,E2 -6197.332} C_VEL
LIN {X 0,Y 496.515,Z 277.333,A -85,B 0,C 180,E1 -6198.158,E2 -6198.158} C_VEL
LIN {X 0,Y 496.19,Z 286.266,A -85,B 0,C 180,E1 -6198.978,E2 -6198.978} C_VEL
LIN {X 0,Y 495.796,Z 295.438,A -85,B 0,C 180,E1 -6200.001,E2 -6200.001} C_VEL
LIN {X 0,Y 495.519,Z 304.378,A -85,B 0,C 180,E1 -6201.231,E2 -6201.231} C_VEL
LIN {X 0,Y 495.277,Z 311.573,A -85,B 0,C 180,E1 -6202.459,E2 -6202.459} C_VEL
LIN {X 0,Y 495.123,Z 317.614,A -85,B 0,C 180,E1 -6203.761,E2 -6203.761} C_VEL
LIN {X 0,Y 495.036,Z 322.461,A -85,B 0,C 180,E1 -6205.114,E2 -6205.114} C_VEL
LIN {X 0,Y 495.031,Z 324.756,A -85,B 0,C 180,E1 -6205.93,E2 -6205.93} C_VEL
LIN {X 0,Y 495.041,Z 326.617,A -85,B 0,C 180,E1 -6206.745,E2 -6206.745} C_VEL
LIN {X 0,Y 494.998,Z 328.011,A -85,B 0,C 180,E1 -6207.56,E2 -6207.56} C_VEL
LIN {X 0,Y 494.962,Z 329.005,A -85,B 0,C 180,E1 -6208.373,E2 -6208.373} C_VEL
LIN {X 0,Y 494.899,Z 329.826,A -85,B 0,C 180,E1 -6210.001,E2 -6210.001} C_VEL
LIN {X 0,Y 494.962,Z 329.004,A -85,B 0,C 180,E1 -6211.628,E2 -6211.628} C_VEL
LIN {X 0,Y 494.998,Z 328.01,A -85,B 0,C 180,E1 -6212.442,E2 -6212.442} C_VEL
LIN {X 0,Y 495.042,Z 326.615,A -85,B 0,C 180,E1 -6213.256,E2 -6213.256} C_VEL
LIN {X 0,Y 495.007,Z 323.679,A -85,B 0,C 180,E1 -6214.479,E2 -6214.479} C_VEL
LIN {X 0,Y 495.125,Z 319.708,A -85,B 0,C 180,E1 -6215.702,E2 -6215.702} C_VEL
LIN {X 0,Y 495.256,Z 313.599,A -85,B 0,C 180,E1 -6217.133,E2 -6217.133} C_VEL
LIN {X 0,Y 495.428,Z 306.923,A -85,B 0,C 180,E1 -6218.361,E2 -6218.361} C_VEL
LIN {X 0,Y 495.704,Z 298.641,A -85,B 0,C 180,E1 -6219.589,E2 -6219.589} C_VEL
LIN {X 0,Y 495.989,Z 290.153,A -85,B 0,C 180,E1 -6220.615,E2 -6220.615} C_VEL
LIN {X 0,Y 496.385,Z 279.668,A -85,B 0,C 180,E1 -6221.639,E2 -6221.639} C_VEL
LIN {X 0,Y 496.743,Z 268.484,A -85,B 0,C 180,E1 -6222.519,E2 -6222.519} C_VEL
LIN {X 0,Y 497.091,Z 257.931,A -85,B 0,C 180,E1 -6223.178,E2 -6223.178} C_VEL
LIN {X 0,Y 497.501,Z 246.288,A -85,B 0,C 180,E1 -6223.739,E2 -6223.739} C_VEL
LIN {X 0,Y 497.459,Z 237.585,A -85,B 0,C 180,E1 -6224.066,E2 -6224.066} C_VEL
LIN {X 0,Y 495.335,Z 224.195,A -85,B 0,C 180,E1 -6224.481,E2 -6224.481} C_VEL
LIN {X 0,Y 495.189,Z 222.953,A -85,B 0,C 180,E1 -6224.538,E2 -6224.538} C_VEL
LIN {X 0,Y 495.324,Z 215.644,A -85,B 0,C 180,E1 -6227.335,E2 -6227.335} C_VEL
LIN {X 0,Y 495.48,Z 207.316,A -85,B 0,C 180,E1 -6230.584,E2 -6230.584} C_VEL
LIN {X 0,Y 495.691,Z 199.066,A -85,B 0,C 180,E1 -6233.832,E2 -6233.832} C_VEL
LIN {X 0,Y 495.864,Z 191.839,A -85,B 0,C 180,E1 -6236.758,E2 -6236.758} C_VEL
LIN {X 0,Y 496.138,Z 184.74,A -85,B 0,C 180,E1 -6239.72,E2 -6239.72} C_VEL
LIN {X 0,Y 496.366,Z 178.176,A -85,B 0,C 180,E1 -6242.548,E2 -6242.548} C_VEL
LIN {X 0,Y 496.575,Z 171.677,A -85,B 0,C 180,E1 -6245.467,E2 -6245.467} C_VEL
LIN {X 0,Y 495.86,Z 166.325,A -85,B 0,C 180,E1 -6248.061,E2 -6248.061} C_VEL
LIN {X 0,Y 495.77,Z 165.736,A -85,B 0,C 180,E1 -6248.457,E2 -6248.457} C_VEL
LIN {X 0,Y 495.766,Z 165.733,A -85,B 0,C 180,E1 -6251.777,E2 -6251.777} C_VEL
LIN {X 0,Y 495.735,Z 165.736,A -85,B 0,C 180,E1 -6255.138,E2 -6255.138} C_VEL
LIN {X 0,Y 495.74,Z 165.735,A -85,B 0,C 180,E1 -6258.217,E2 -6258.217} C_VEL
LIN {X 0,Y 495.732,Z 165.735,A -85,B 0,C 180,E1 -6261.407,E2 -6261.407} C_VEL
LIN {X 0,Y 495.739,Z 165.731,A -85,B 0,C 180,E1 -6264.462,E2 -6264.462} C_VEL
LIN {X 0,Y 495.749,Z 165.733,A -85,B 0,C 180,E1 -6267.404,E2 -6267.404} C_VEL
LIN {X 0,Y 495.746,Z 165.733,A -85,B 0,C 180,E1 -6270.252,E2 -6270.252} C_VEL
LIN {X 0,Y 495.8,Z 165.727,A -85,B 0,C 180,E1 -6273.249,E2 -6273.249} C_VEL
LIN {X 0,Y 495.746,Z 165.733,A -85,B 0,C 180,E1 -6275.725,E2 -6275.725} C_VEL
LIN {X 0,Y 495.741,Z 165.732,A -85,B 0,C 180,E1 -6278.371,E2 -6278.371} C_VEL
LIN {X 0,Y 495.805,Z 165.726,A -85,B 0,C 180,E1 -6281.743,E2 -6281.743} C_VEL
LIN {X 0,Y 495.796,Z 165.726,A -85,B 0,C 180,E1 -6284.547,E2 -6284.547} C_VEL
LIN {X 0,Y 495.851,Z 165.719,A -85,B 0,C 180,E1 -6287.937,E2 -6287.937} C_VEL
LIN {X 0,Y 495.837,Z 165.72,A -85,B 0,C 180,E1 -6291.03,E2 -6291.03} C_VEL
LIN {X 0,Y 495.886,Z 165.715,A -85,B 0,C 180,E1 -6293.49,E2 -6293.49} C_VEL
LIN {X 0,Y 495.819,Z 165.724,A -85,B 0,C 180,E1 -6296.75,E2 -6296.75} C_VEL
LIN {X 0,Y 495.953,Z 165.708,A -85,B 0,C 180,E1 -6299.188,E2 -6299.188} C_VEL
LIN {X 0,Y 495.842,Z 165.719,A -85,B 0,C 180,E1 -6301.625,E2 -6301.625} C_VEL
LIN {X 0,Y 495.848,Z 165.717,A -85,B 0,C 180,E1 -6303.25,E2 -6303.25} C_VEL
LIN {X 0,Y 495.856,Z 165.718,A -85,B 0,C 180,E1 -6306.511,E2 -6306.511} C_VEL
LIN {X 0,Y 495.817,Z 165.725,A -85,B 0,C 180,E1 -6308.97,E2 -6308.97} C_VEL
LIN {X 0,Y 495.8,Z 165.727,A -85,B 0,C 180,E1 -6312.036,E2 -6312.036} C_VEL
LIN {X 0,Y 495.798,Z 165.726,A -85,B 0,C 180,E1 -6315.453,E2 -6315.453} C_VEL
LIN {X 0,Y 495.806,Z 165.723,A -85,B 0,C 180,E1 -6318.257,E2 -6318.257} C_VEL
LIN {X 0,Y 495.732,Z 165.734,A -85,B 0,C 180,E1 -6321.63,E2 -6321.63} C_VEL
LIN {X 0,Y 495.756,Z 165.731,A -85,B 0,C 180,E1 -6324.875,E2 -6324.875} C_VEL
LIN {X 0,Y 495.792,Z 165.726,A -85,B 0,C 180,E1 -6326.976,E2 -6326.976} C_VEL
LIN {X 0,Y 495.756,Z 165.729,A -85,B 0,C 180,E1 -6330.151,E2 -6330.151} C_VEL
LIN {X 0,Y 495.775,Z 165.729,A -85,B 0,C 180,E1 -6333.246,E2 -6333.246} C_VEL
LIN {X 0,Y 495.708,Z 165.738,A -85,B 0,C 180,E1 -6336.091,E2 -6336.091} C_VEL
LIN {X 0,Y 495.747,Z 165.732,A -85,B 0,C 180,E1 -6338.77,E2 -6338.77} C_VEL
LIN {X 0,Y 495.744,Z 165.73,A -85,B 0,C 180,E1 -6341.783,E2 -6341.783} C_VEL
LIN {X 0,Y 495.738,Z 165.733,A -85,B 0,C 180,E1 -6345.141,E2 -6345.141} C_VEL
LIN {X 0,Y 495.746,Z 165.734,A -85,B 0,C 180,E1 -6348.221,E2 -6348.221} C_VEL
LIN {X 0,Y 495.724,Z 165.74,A -85,B 0,C 180,E1 -6351.238,E2 -6351.238} C_VEL
LIN {X 0,Y 495.613,Z 165.776,A -85,B 0,C 180,E1 -6352.571,E2 -6352.571} C_VEL
LIN {X 0,Y 495.619,Z 169.87,A -85,B 0,C 180,E1 -6355.446,E2 -6355.446} C_VEL
LIN {X 0,Y 495.542,Z 174.132,A -85,B 0,C 180,E1 -6358.35,E2 -6358.35} C_VEL
LIN {X 0,Y 495.453,Z 177.557,A -85,B 0,C 180,E1 -6360.639,E2 -6360.639} C_VEL
LIN {X 0,Y 494.752,Z 178.642,A -85,B 0,C 180,E1 -6361.305,E2 -6361.305} C_VEL
LIN {X 0,Y 491.838,Z 180.581,A -85,B 0,C 180,E1 -6362.383,E2 -6362.383} C_VEL
LIN {X 0,Y 489.389,Z 182.151,A -85,B 0,C 180,E1 -6363.251,E2 -6363.251} C_VEL
LIN {X 0,Y 488.342,Z 183.281,A -85,B 0,C 180,E1 -6363.924,E2 -6363.924} C_VEL
LIN {X 0,Y 488.258,Z 183.638,A -85,B 0,C 180,E1 -6364.152,E2 -6364.152} C_VEL
LIN {X 0,Y 488.212,Z 188.216,A -85,B 0,C 180,E1 -6367.119,E2 -6367.119} C_VEL
LIN {X 0,Y 488.104,Z 193.909,A -85,B 0,C 180,E1 -6370.661,E2 -6370.661} C_VEL
LIN {X 0,Y 488.024,Z 198.269,A -85,B 0,C 180,E1 -6373.335,E2 -6373.335} C_VEL
LIN {X 0,Y 490.869,Z 212.669,A -85,B 0,C 180,E1 -6373.842,E2 -6373.842} C_VEL
LIN {X 0,Y 490.601,Z 225.257,A -85,B 0,C 180,E1 -6374.366,E2 -6374.366} C_VEL
LIN {X 0,Y 490.179,Z 237.212,A -85,B 0,C 180,E1 -6375.045,E2 -6375.045} C_VEL
LIN {X 0,Y 489.706,Z 248.644,A -85,B 0,C 180,E1 -6375.879,E2 -6375.879} C_VEL
LIN {X 0,Y 489.389,Z 258.934,A -85,B 0,C 180,E1 -6376.822,E2 -6376.822} C_VEL
LIN {X 0,Y 488.942,Z 268.913,A -85,B 0,C 180,E1 -6377.964,E2 -6377.964} C_VEL
LIN {X 0,Y 488.698,Z 277.771,A -85,B 0,C 180,E1 -6379.225,E2 -6379.225} C_VEL
LIN {X 0,Y 488.388,Z 284.808,A -85,B 0,C 180,E1 -6380.475,E2 -6380.475} C_VEL
LIN {X 0,Y 488.193,Z 290.415,A -85,B 0,C 180,E1 -6381.723,E2 -6381.723} C_VEL
LIN {X 0,Y 488.073,Z 294.821,A -85,B 0,C 180,E1 -6382.97,E2 -6382.97} C_VEL
LIN {X 0,Y 488,Z 298.155,A -85,B 0,C 180,E1 -6384.214,E2 -6384.214} C_VEL
LIN {X 0,Y 487.924,Z 301.064,A -85,B 0,C 180,E1 -6385.87,E2 -6385.87} C_VEL
LIN {X 0,Y 487.957,Z 301.924,A -85,B 0,C 180,E1 -6386.697,E2 -6386.697} C_VEL
LIN {X 0,Y 487.891,Z 302.396,A -85,B 0,C 180,E1 -6388.349,E2 -6388.349} C_VEL
LIN {X 0,Y 487.825,Z 301.343,A -85,B 0,C 180,E1 -6389.999,E2 -6389.999} C_VEL
LIN {X 0,Y 487.843,Z 300.194,A -85,B 0,C 180,E1 -6390.825,E2 -6390.825} C_VEL
LIN {X 0,Y 487.922,Z 298.633,A -85,B 0,C 180,E1 -6391.65,E2 -6391.65} C_VEL
LIN {X 0,Y 488.091,Z 295.501,A -85,B 0,C 180,E1 -6392.888,E2 -6392.888} C_VEL
LIN {X 0,Y 488.193,Z 291.326,A -85,B 0,C 180,E1 -6394.127,E2 -6394.127} C_VEL
LIN {X 0,Y 488.373,Z 284.985,A -85,B 0,C 180,E1 -6395.573,E2 -6395.573} C_VEL
LIN {X 0,Y 488.696,Z 277.913,A -85,B 0,C 180,E1 -6396.836,E2 -6396.836} C_VEL
LIN {X 0,Y 488.927,Z 269.4,A -85,B 0,C 180,E1 -6398.055,E2 -6398.055} C_VEL
LIN {X 0,Y 489.345,Z 260.525,A -85,B 0,C 180,E1 -6399.089,E2 -6399.089} C_VEL
LIN {X 0,Y 489.75,Z 250.77,A -85,B 0,C 180,E1 -6400.019,E2 -6400.019} C_VEL
LIN {X 0,Y 490.084,Z 240.015,A -85,B 0,C 180,E1 -6400.847,E2 -6400.847} C_VEL
LIN {X 0,Y 490.433,Z 227.955,A -85,B 0,C 180,E1 -6401.572,E2 -6401.572} C_VEL
LIN {X 0,Y 490.835,Z 215.349,A -85,B 0,C 180,E1 -6402.138,E2 -6402.138} C_VEL
LIN {X 0,Y 490.562,Z 210.49,A -85,B 0,C 180,E1 -6402.318,E2 -6402.318} C_VEL
LIN {X 0,Y 488.061,Z 198.254,A -85,B 0,C 180,E1 -6402.734,E2 -6402.734} C_VEL
LIN {X 0,Y 488.119,Z 193.107,A -85,B 0,C 180,E1 -6405.875,E2 -6405.875} C_VEL
LIN {X 0,Y 488.164,Z 188.914,A -85,B 0,C 180,E1 -6408.463,E2 -6408.463} C_VEL
LIN {X 0,Y 488.261,Z 184.785,A -85,B 0,C 180,E1 -6411.089,E2 -6411.089} C_VEL
LIN {X 0,Y 488.312,Z 180.684,A -85,B 0,C 180,E1 -6413.763,E2 -6413.763} C_VEL
LIN {X 0,Y 488.407,Z 176.009,A -85,B 0,C 180,E1 -6416.853,E2 -6416.853} C_VEL
LIN {X 0,Y 488.504,Z 172.394,A -85,B 0,C 180,E1 -6419.282,E2 -6419.282} C_VEL
LIN {X 0,Y 488.574,Z 168.221,A -85,B 0,C 180,E1 -6422.153,E2 -6422.153} C_VEL
LIN {X 0,Y 488.576,Z 166.632,A -85,B 0,C 180,E1 -6423.455,E2 -6423.455} C_VEL
LIN {X 0,Y 488.696,Z 166.614,A -85,B 0,C 180,E1 -6425.113,E2 -6425.113} C_VEL
LIN {X 0,Y 488.663,Z 166.617,A -85,B 0,C 180,E1 -6428.198,E2 -6428.198} C_VEL
LIN {X 0,Y 488.704,Z 166.611,A -85,B 0,C 180,E1 -6430.342,E2 -6430.342} C_VEL
LIN {X 0,Y 488.699,Z 166.609,A -85,B 0,C 180,E1 -6432.824,E2 -6432.824} C_VEL
LIN {X 0,Y 488.683,Z 166.611,A -85,B 0,C 180,E1 -6435.973,E2 -6435.973} C_VEL
LIN {X 0,Y 488.706,Z 166.609,A -85,B 0,C 180,E1 -6438.584,E2 -6438.584} C_VEL
LIN {X 0,Y 488.718,Z 166.61,A -85,B 0,C 180,E1 -6440.939,E2 -6440.939} C_VEL
LIN {X 0,Y 488.654,Z 166.617,A -85,B 0,C 180,E1 -6443.865,E2 -6443.865} C_VEL
LIN {X 0,Y 488.712,Z 166.608,A -85,B 0,C 180,E1 -6446.875,E2 -6446.875} C_VEL
LIN {X 0,Y 488.706,Z 166.61,A -85,B 0,C 180,E1 -6449.779,E2 -6449.779} C_VEL
LIN {X 0,Y 488.769,Z 166.603,A -85,B 0,C 180,E1 -6453.052,E2 -6453.052} C_VEL
LIN {X 0,Y 488.687,Z 166.613,A -85,B 0,C 180,E1 -6456.254,E2 -6456.254} C_VEL
LIN {X 0,Y 488.714,Z 166.607,A -85,B 0,C 180,E1 -6459.173,E2 -6459.173} C_VEL
LIN {X 0,Y 488.701,Z 166.61,A -85,B 0,C 180,E1 -6462.422,E2 -6462.422} C_VEL
LIN {X 0,Y 488.732,Z 166.608,A -85,B 0,C 180,E1 -6464.998,E2 -6464.998} C_VEL
LIN {X 0,Y 488.815,Z 166.599,A -85,B 0,C 180,E1 -6468.388,E2 -6468.388} C_VEL
LIN {X 0,Y 488.825,Z 166.595,A -85,B 0,C 180,E1 -6471.734,E2 -6471.734} C_VEL
LIN {X 0,Y 488.852,Z 166.591,A -85,B 0,C 180,E1 -6474.224,E2 -6474.224} C_VEL
LIN {X 0,Y 488.923,Z 166.586,A -85,B 0,C 180,E1 -6477.528,E2 -6477.528} C_VEL
LIN {X 0,Y 488.939,Z 166.582,A -85,B 0,C 180,E1 -6480.823,E2 -6480.823} C_VEL
LIN {X 0,Y 488.783,Z 166.599,A -85,B 0,C 180,E1 -6483.297,E2 -6483.297} C_VEL
LIN {X 0,Y 488.816,Z 166.595,A -85,B 0,C 180,E1 -6486.605,E2 -6486.605} C_VEL
LIN {X 0,Y 488.772,Z 166.601,A -85,B 0,C 180,E1 -6489.1,E2 -6489.1} C_VEL
LIN {X 0,Y 488.788,Z 166.597,A -85,B 0,C 180,E1 -6492.136,E2 -6492.136} C_VEL
LIN {X 0,Y 488.74,Z 166.605,A -85,B 0,C 180,E1 -6495.556,E2 -6495.556} C_VEL
LIN {X 0,Y 488.719,Z 166.61,A -85,B 0,C 180,E1 -6498.443,E2 -6498.443} C_VEL
LIN {X 0,Y 488.708,Z 166.609,A -85,B 0,C 180,E1 -6501.071,E2 -6501.071} C_VEL
LIN {X 0,Y 488.685,Z 166.612,A -85,B 0,C 180,E1 -6503.746,E2 -6503.746} C_VEL
LIN {X 0,Y 488.768,Z 166.606,A -85,B 0,C 180,E1 -6506.947,E2 -6506.947} C_VEL
LIN {X 0,Y 488.689,Z 166.613,A -85,B 0,C 180,E1 -6510.367,E2 -6510.367} C_VEL
LIN {X 0,Y 488.707,Z 166.61,A -85,B 0,C 180,E1 -6513.486,E2 -6513.486} C_VEL
LIN {X 0,Y 488.661,Z 166.615,A -85,B 0,C 180,E1 -6516.358,E2 -6516.358} C_VEL
LIN {X 0,Y 488.725,Z 166.608,A -85,B 0,C 180,E1 -6519.252,E2 -6519.252} C_VEL
LIN {X 0,Y 488.712,Z 166.612,A -85,B 0,C 180,E1 -6522.523,E2 -6522.523} C_VEL
LIN {X 0,Y 488.692,Z 166.608,A -85,B 0,C 180,E1 -6525.201,E2 -6525.201} C_VEL
LIN {X 0,Y 488.712,Z 166.612,A -85,B 0,C 180,E1 -6527.481,E2 -6527.481} C_VEL
LIN {X 0,Y 488.683,Z 166.615,A -85,B 0,C 180,E1 -6530.748,E2 -6530.748} C_VEL
LIN {X 0,Y 488.721,Z 166.722,A -85,B 0,C 180,E1 -6531.808,E2 -6531.808} C_VEL
LIN {X 0,Y 489.507,Z 172.197,A -85,B 0,C 180,E1 -6534.45,E2 -6534.45} C_VEL
LIN {X 0,Y 489.322,Z 177.702,A -85,B 0,C 180,E1 -6536.925,E2 -6536.925} C_VEL
LIN {X 0,Y 489.146,Z 184.327,A -85,B 0,C 180,E1 -6539.813,E2 -6539.813} C_VEL
LIN {X 0,Y 488.846,Z 191.004,A -85,B 0,C 180,E1 -6542.612,E2 -6542.612} C_VEL
LIN {X 0,Y 488.663,Z 197.695,A -85,B 0,C 180,E1 -6545.352,E2 -6545.352} C_VEL
LIN {X 0,Y 488.499,Z 205.499,A -85,B 0,C 180,E1 -6548.48,E2 -6548.48} C_VEL
LIN {X 0,Y 488.3,Z 213.904,A -85,B 0,C 180,E1 -6551.792,E2 -6551.792} C_VEL
LIN {X 0,Y 488.132,Z 222.088,A -85,B 0,C 180,E1 -6554.982,E2 -6554.982} C_VEL
LIN {X 0,Y 488.129,Z 222.845,A -85,B 0,C 180,E1 -6555.275,E2 -6555.275} C_VEL
LIN {X 0,Y 490.372,Z 237.609,A -85,B 0,C 180,E1 -6555.741,E2 -6555.741} C_VEL
LIN {X 0,Y 490.723,Z 240.688,A -85,B 0,C 180,E1 -6555.857,E2 -6555.857} C_VEL
LIN {X 0,Y 490.333,Z 252.763,A -85,B 0,C 180,E1 -6556.375,E2 -6556.375} C_VEL
LIN {X 0,Y 489.907,Z 264.979,A -85,B 0,C 180,E1 -6557.08,E2 -6557.08} C_VEL
LIN {X 0,Y 489.578,Z 275.835,A -85,B 0,C 180,E1 -6557.882,E2 -6557.882} C_VEL
LIN {X 0,Y 489.198,Z 286.046,A -85,B 0,C 180,E1 -6558.818,E2 -6558.818} C_VEL
LIN {X 0,Y 488.752,Z 295.226,A -85,B 0,C 180,E1 -6559.856,E2 -6559.856} C_VEL
LIN {X 0,Y 488.456,Z 304.173,A -85,B 0,C 180,E1 -6561.103,E2 -6561.103} C_VEL
LIN {X 0,Y 488.21,Z 311.372,A -85,B 0,C 180,E1 -6562.349,E2 -6562.349} C_VEL
LIN {X 0,Y 488.023,Z 317.894,A -85,B 0,C 180,E1 -6563.792,E2 -6563.792} C_VEL
LIN {X 0,Y 487.967,Z 322.263,A -85,B 0,C 180,E1 -6565.043,E2 -6565.043} C_VEL
LIN {X 0,Y 487.927,Z 324.558,A -85,B 0,C 180,E1 -6565.871,E2 -6565.871} C_VEL
LIN {X 0,Y 487.964,Z 326.42,A -85,B 0,C 180,E1 -6566.698,E2 -6566.698} C_VEL
LIN {X 0,Y 487.891,Z 328.808,A -85,B 0,C 180,E1 -6568.35,E2 -6568.35} C_VEL
LIN {X 0,Y 487.82,Z 329.629,A -85,B 0,C 180,E1 -6570.001,E2 -6570.001} C_VEL
LIN {X 0,Y 487.891,Z 328.807,A -85,B 0,C 180,E1 -6571.651,E2 -6571.651} C_VEL
LIN {X 0,Y 487.964,Z 326.417,A -85,B 0,C 180,E1 -6573.303,E2 -6573.303} C_VEL
LIN {X 0,Y 487.92,Z 323.48,A -85,B 0,C 180,E1 -6574.544,E2 -6574.544} C_VEL
LIN {X 0,Y 488.022,Z 319.509,A -85,B 0,C 180,E1 -6575.786,E2 -6575.786} C_VEL
LIN {X 0,Y 488.181,Z 313.402,A -85,B 0,C 180,E1 -6577.237,E2 -6577.237} C_VEL
LIN {X 0,Y 488.362,Z 306.729,A -85,B 0,C 180,E1 -6578.482,E2 -6578.482} C_VEL
LIN {X 0,Y 488.669,Z 298.453,A -85,B 0,C 180,E1 -6579.729,E2 -6579.729} C_VEL
LIN {X 0,Y 488.994,Z 289.974,A -85,B 0,C 180,E1 -6580.768,E2 -6580.768} C_VEL
LIN {X 0,Y 489.419,Z 279.503,A -85,B 0,C 180,E1 -6581.807,E2 -6581.807} C_VEL
LIN {X 0,Y 489.797,Z 268.274,A -85,B 0,C 180,E1 -6582.704,E2 -6582.704} C_VEL
LIN {X 0,Y 490.182,Z 257.801,A -85,B 0,C 180,E1 -6583.367,E2 -6583.367} C_VEL
LIN {X 0,Y 490.611,Z 246.198,A -85,B 0,C 180,E1 -6583.936,E2 -6583.936} C_VEL
LIN {X 0,Y 490.582,Z 238.665,A -85,B 0,C 180,E1 -6584.227,E2 -6584.227} C_VEL
LIN {X 0,Y 488.475,Z 224.95,A -85,B 0,C 180,E1 -6584.676,E2 -6584.676} C_VEL
LIN {X 0,Y 488.124,Z 222.776,A -85,B 0,C 180,E1 -6584.753,E2 -6584.753} C_VEL
LIN {X 0,Y 488.253,Z 215.497,A -85,B 0,C 180,E1 -6587.594,E2 -6587.594} C_VEL
LIN {X 0,Y 488.449,Z 207.593,A -85,B 0,C 180,E1 -6590.732,E2 -6590.732} C_VEL
LIN {X 0,Y 488.642,Z 200.067,A -85,B 0,C 180,E1 -6593.747,E2 -6593.747} C_VEL
LIN {X 0,Y 488.798,Z 193.452,A -85,B 0,C 180,E1 -6596.468,E2 -6596.468} C_VEL
LIN {X 0,Y 489.106,Z 186.861,A -85,B 0,C 180,E1 -6599.244,E2 -6599.244} C_VEL
LIN {X 0,Y 489.358,Z 179.209,A -85,B 0,C 180,E1 -6602.584,E2 -6602.584} C_VEL
LIN {X 0,Y 489.56,Z 172.721,A -85,B 0,C 180,E1 -6605.547,E2 -6605.547} C_VEL
LIN {X 0,Y 488.967,Z 168.197,A -85,B 0,C 180,E1 -6607.765,E2 -6607.765} C_VEL
LIN {X 0,Y 488.711,Z 166.616,A -85,B 0,C 180,E1 -6608.589,E2 -6608.589} C_VEL
LIN {X 0,Y 488.712,Z 166.61,A -85,B 0,C 180,E1 -6611.6,E2 -6611.6} C_VEL
LIN {X 0,Y 488.689,Z 166.612,A -85,B 0,C 180,E1 -6614.022,E2 -6614.022} C_VEL
LIN {X 0,Y 488.694,Z 166.614,A -85,B 0,C 180,E1 -6617.172,E2 -6617.172} C_VEL
LIN {X 0,Y 488.717,Z 166.609,A -85,B 0,C 180,E1 -6619.675,E2 -6619.675} C_VEL
LIN {X 0,Y 488.664,Z 166.614,A -85,B 0,C 180,E1 -6622.84,E2 -6622.84} C_VEL
LIN {X 0,Y 488.716,Z 166.607,A -85,B 0,C 180,E1 -6625.886,E2 -6625.886} C_VEL
LIN {X 0,Y 488.673,Z 166.616,A -85,B 0,C 180,E1 -6628.819,E2 -6628.819} C_VEL
LIN {X 0,Y 488.722,Z 166.609,A -85,B 0,C 180,E1 -6631.67,E2 -6631.67} C_VEL
LIN {X 0,Y 488.726,Z 166.607,A -85,B 0,C 180,E1 -6634.443,E2 -6634.443} C_VEL
LIN {X 0,Y 488.726,Z 166.61,A -85,B 0,C 180,E1 -6637.153,E2 -6637.153} C_VEL
LIN {X 0,Y 488.704,Z 166.608,A -85,B 0,C 180,E1 -6639.81,E2 -6639.81} C_VEL
LIN {X 0,Y 488.722,Z 166.611,A -85,B 0,C 180,E1 -6642.423,E2 -6642.423} C_VEL
LIN {X 0,Y 488.733,Z 166.607,A -85,B 0,C 180,E1 -6644.999,E2 -6644.999} C_VEL
LIN {X 0,Y 488.811,Z 166.596,A -85,B 0,C 180,E1 -6648.388,E2 -6648.388} C_VEL
LIN {X 0,Y 488.821,Z 166.593,A -85,B 0,C 180,E1 -6651.734,E2 -6651.734} C_VEL
LIN {X 0,Y 488.861,Z 166.593,A -85,B 0,C 180,E1 -6654.224,E2 -6654.224} C_VEL
LIN {X 0,Y 488.93,Z 166.583,A -85,B 0,C 180,E1 -6657.529,E2 -6657.529} C_VEL
LIN {X 0,Y 488.948,Z 166.58,A -85,B 0,C 180,E1 -6660.824,E2 -6660.824} C_VEL
LIN {X 0,Y 488.792,Z 166.596,A -85,B 0,C 180,E1 -6663.297,E2 -6663.297} C_VEL
LIN {X 0,Y 488.848,Z 166.595,A -85,B 0,C 180,E1 -6665.776,E2 -6665.776} C_VEL
LIN {X 0,Y 488.79,Z 166.599,A -85,B 0,C 180,E1 -6668.267,E2 -6668.267} C_VEL
LIN {X 0,Y 488.778,Z 166.601,A -85,B 0,C 180,E1 -6671.613,E2 -6671.613} C_VEL
LIN {X 0,Y 488.735,Z 166.604,A -85,B 0,C 180,E1 -6675.002,E2 -6675.002} C_VEL
LIN {X 0,Y 488.742,Z 166.603,A -85,B 0,C 180,E1 -6678.443,E2 -6678.443} C_VEL
LIN {X 0,Y 488.687,Z 166.615,A -85,B 0,C 180,E1 -6681.072,E2 -6681.072} C_VEL
LIN {X 0,Y 488.672,Z 166.615,A -85,B 0,C 180,E1 -6683.747,E2 -6683.747} C_VEL
LIN {X 0,Y 488.77,Z 166.601,A -85,B 0,C 180,E1 -6686.945,E2 -6686.945} C_VEL
LIN {X 0,Y 488.714,Z 166.606,A -85,B 0,C 180,E1 -6690.22,E2 -6690.22} C_VEL
LIN {X 0,Y 488.717,Z 166.608,A -85,B 0,C 180,E1 -6693.486,E2 -6693.486} C_VEL
LIN {X 0,Y 488.669,Z 166.616,A -85,B 0,C 180,E1 -6696.357,E2 -6696.357} C_VEL
LIN {X 0,Y 488.685,Z 166.615,A -85,B 0,C 180,E1 -6699.256,E2 -6699.256} C_VEL
LIN {X 0,Y 488.694,Z 166.609,A -85,B 0,C 180,E1 -6701.602,E2 -6701.602} C_VEL
LIN {X 0,Y 488.7,Z 166.611,A -85,B 0,C 180,E1 -6704.803,E2 -6704.803} C_VEL
LIN {X 0,Y 488.681,Z 166.614,A -85,B 0,C 180,E1 -6707.476,E2 -6707.476} C_VEL
LIN {X 0,Y 488.725,Z 166.608,A -85,B 0,C 180,E1 -6709.679,E2 -6709.679} C_VEL
LIN {X 0,Y 488.597,Z 166.625,A -85,B 0,C 180,E1 -6712.291,E2 -6712.291} C_VEL
LIN {X 0,Y 488.59,Z 168.217,A -85,B 0,C 180,E1 -6713.661,E2 -6713.661} C_VEL
LIN {X 0,Y 488.555,Z 172.325,A -85,B 0,C 180,E1 -6716.549,E2 -6716.549} C_VEL
LIN {X 0,Y 488.441,Z 177.028,A -85,B 0,C 180,E1 -6719.763,E2 -6719.763} C_VEL
LIN {X 0,Y 488.326,Z 181.25,A -85,B 0,C 180,E1 -6722.579,E2 -6722.579} C_VEL
LIN {X 0,Y 488.258,Z 183.638,A -85,B 0,C 180,E1 -6724.152,E2 -6724.152} C_VEL
LIN {X 0,Y 487.593,Z 184.741,A -85,B 0,C 180,E1 -6724.828,E2 -6724.828} C_VEL
LIN {X 0,Y 484.717,Z 186.699,A -85,B 0,C 180,E1 -6725.921,E2 -6725.921} C_VEL
LIN {X 0,Y 482.261,Z 188.293,A -85,B 0,C 180,E1 -6726.801,E2 -6726.801} C_VEL
LIN {X 0,Y 481.178,Z 189.457,A -85,B 0,C 180,E1 -6727.482,E2 -6727.482} C_VEL
LIN {X 0,Y 481.075,Z 189.831,A -85,B 0,C 180,E1 -6727.714,E2 -6727.714} C_VEL
LIN {X 0,Y 481.024,Z 194.048,A -85,B 0,C 180,E1 -6730.365,E2 -6730.365} C_VEL
LIN {X 0,Y 480.96,Z 198.601,A -85,B 0,C 180,E1 -6733.118,E2 -6733.118} C_VEL
LIN {X 0,Y 483.717,Z 211.944,A -85,B 0,C 180,E1 -6733.587,E2 -6733.587} C_VEL
LIN {X 0,Y 483.977,Z 217.477,A -85,B 0,C 180,E1 -6733.806,E2 -6733.806} C_VEL
LIN {X 0,Y 483.663,Z 228.052,A -85,B 0,C 180,E1 -6734.298,E2 -6734.298} C_VEL
LIN {X 0,Y 483.171,Z 240.242,A -85,B 0,C 180,E1 -6735.038,E2 -6735.038} C_VEL
LIN {X 0,Y 482.754,Z 251.077,A -85,B 0,C 180,E1 -6735.887,E2 -6735.887} C_VEL
LIN {X 0,Y 482.305,Z 261.863,A -85,B 0,C 180,E1 -6736.947,E2 -6736.947} C_VEL
LIN {X 0,Y 481.85,Z 270.897,A -85,B 0,C 180,E1 -6738.042,E2 -6738.042} C_VEL
LIN {X 0,Y 481.605,Z 279.102,A -85,B 0,C 180,E1 -6739.277,E2 -6739.277} C_VEL
LIN {X 0,Y 481.3,Z 285.898,A -85,B 0,C 180,E1 -6740.545,E2 -6740.545} C_VEL
LIN {X 0,Y 481.099,Z 292.128,A -85,B 0,C 180,E1 -6742.023,E2 -6742.023} C_VEL
LIN {X 0,Y 480.968,Z 296.843,A -85,B 0,C 180,E1 -6743.534,E2 -6743.534} C_VEL
LIN {X 0,Y 480.846,Z 299.965,A -85,B 0,C 180,E1 -6744.969,E2 -6744.969} C_VEL
LIN {X 0,Y 480.882,Z 302.1,A -85,B 0,C 180,E1 -6746.648,E2 -6746.648} C_VEL
LIN {X 0,Y 480.822,Z 302.598,A -85,B 0,C 180,E1 -6748.324,E2 -6748.324} C_VEL
LIN {X 0,Y 480.749,Z 301.564,A -85,B 0,C 180,E1 -6749.999,E2 -6749.999} C_VEL
LIN {X 0,Y 480.769,Z 300.434,A -85,B 0,C 180,E1 -6750.837,E2 -6750.837} C_VEL
LIN {X 0,Y 480.853,Z 298.882,A -85,B 0,C 180,E1 -6751.674,E2 -6751.674} C_VEL
LIN {X 0,Y 481.031,Z 295.77,A -85,B 0,C 180,E1 -6752.93,E2 -6752.93} C_VEL
LIN {X 0,Y 481.142,Z 291.616,A -85,B 0,C 180,E1 -6754.187,E2 -6754.187} C_VEL
LIN {X 0,Y 481.296,Z 285.298,A -85,B 0,C 180,E1 -6755.656,E2 -6755.656} C_VEL
LIN {X 0,Y 481.656,Z 278.635,A -85,B 0,C 180,E1 -6756.875,E2 -6756.875} C_VEL
LIN {X 0,Y 481.843,Z 271.38,A -85,B 0,C 180,E1 -6757.964,E2 -6757.964} C_VEL
LIN {X 0,Y 482.289,Z 262.87,A -85,B 0,C 180,E1 -6759.011,E2 -6759.011} C_VEL
LIN {X 0,Y 482.738,Z 252.385,A -85,B 0,C 180,E1 -6760.06,E2 -6760.06} C_VEL
LIN {X 0,Y 483.059,Z 241.994,A -85,B 0,C 180,E1 -6760.901,E2 -6760.901} C_VEL
LIN {X 0,Y 483.486,Z 230.541,A -85,B 0,C 180,E1 -6761.634,E2 -6761.634} C_VEL
LIN {X 0,Y 483.913,Z 218.744,A -85,B 0,C 180,E1 -6762.205,E2 -6762.205} C_VEL
LIN {X 0,Y 483.74,Z 211.961,A -85,B 0,C 180,E1 -6762.472,E2 -6762.472} C_VEL
LIN {X 0,Y 480.98,Z 198.438,A -85,B 0,C 180,E1 -6762.949,E2 -6762.949} C_VEL
LIN {X 0,Y 481.068,Z 194.496,A -85,B 0,C 180,E1 -6765.374,E2 -6765.374} C_VEL
LIN {X 0,Y 481.097,Z 189.099,A -85,B 0,C 180,E1 -6768.744,E2 -6768.744} C_VEL
LIN {X 0,Y 481.198,Z 184.965,A -85,B 0,C 180,E1 -6771.413,E2 -6771.413} C_VEL
LIN {X 0,Y 481.285,Z 180.84,A -85,B 0,C 180,E1 -6774.132,E2 -6774.132} C_VEL
LIN {X 0,Y 481.357,Z 176.49,A -85,B 0,C 180,E1 -6777.047,E2 -6777.047} C_VEL
LIN {X 0,Y 481.475,Z 172.531,A -85,B 0,C 180,E1 -6779.752,E2 -6779.752} C_VEL
LIN {X 0,Y 481.502,Z 168.343,A -85,B 0,C 180,E1 -6782.684,E2 -6782.684} C_VEL
LIN {X 0,Y 481.545,Z 167.505,A -85,B 0,C 180,E1 -6783.705,E2 -6783.705} C_VEL
LIN {X 0,Y 481.617,Z 167.492,A -85,B 0,C 180,E1 -6785.708,E2 -6785.708} C_VEL
LIN {X 0,Y 481.656,Z 167.49,A -85,B 0,C 180,E1 -6788.856,E2 -6788.856} C_VEL
LIN {X 0,Y 481.647,Z 167.491,A -85,B 0,C 180,E1 -6791.911,E2 -6791.911} C_VEL
LIN {X 0,Y 481.643,Z 167.488,A -85,B 0,C 180,E1 -6794.454,E2 -6794.454} C_VEL
LIN {X 0,Y 481.67,Z 167.486,A -85,B 0,C 180,E1 -6796.843,E2 -6796.843} C_VEL
LIN {X 0,Y 481.668,Z 167.485,A -85,B 0,C 180,E1 -6800.058,E2 -6800.058} C_VEL
LIN {X 0,Y 481.602,Z 167.494,A -85,B 0,C 180,E1 -6803.25,E2 -6803.25} C_VEL
LIN {X 0,Y 481.684,Z 167.486,A -85,B 0,C 180,E1 -6806.328,E2 -6806.328} C_VEL
LIN {X 0,Y 481.631,Z 167.492,A -85,B 0,C 180,E1 -6809.413,E2 -6809.413} C_VEL
LIN {X 0,Y 481.675,Z 167.484,A -85,B 0,C 180,E1 -6812.166,E2 -6812.166} C_VEL
LIN {X 0,Y 481.705,Z 167.481,A -85,B 0,C 180,E1 -6814.969,E2 -6814.969} C_VEL
LIN {X 0,Y 481.643,Z 167.488,A -85,B 0,C 180,E1 -6817.704,E2 -6817.704} C_VEL
LIN {X 0,Y 481.673,Z 167.486,A -85,B 0,C 180,E1 -6820.391,E2 -6820.391} C_VEL
LIN {X 0,Y 481.659,Z 167.489,A -85,B 0,C 180,E1 -6823.032,E2 -6823.032} C_VEL
LIN {X 0,Y 481.667,Z 167.487,A -85,B 0,C 180,E1 -6825.638,E2 -6825.638} C_VEL
LIN {X 0,Y 481.773,Z 167.475,A -85,B 0,C 180,E1 -6828.215,E2 -6828.215} C_VEL
LIN {X 0,Y 481.766,Z 167.473,A -85,B 0,C 180,E1 -6831.612,E2 -6831.612} C_VEL
LIN {X 0,Y 481.812,Z 167.469,A -85,B 0,C 180,E1 -6834.139,E2 -6834.139} C_VEL
LIN {X 0,Y 481.89,Z 167.462,A -85,B 0,C 180,E1 -6837.492,E2 -6837.492} C_VEL
LIN {X 0,Y 481.889,Z 167.46,A -85,B 0,C 180,E1 -6840.835,E2 -6840.835} C_VEL
LIN {X 0,Y 481.899,Z 167.459,A -85,B 0,C 180,E1 -6842.507,E2 -6842.507} C_VEL
LIN {X 0,Y 481.807,Z 167.473,A -85,B 0,C 180,E1 -6845.86,E2 -6845.86} C_VEL
LIN {X 0,Y 481.765,Z 167.472,A -85,B 0,C 180,E1 -6848.388,E2 -6848.388} C_VEL
LIN {X 0,Y 481.765,Z 167.473,A -85,B 0,C 180,E1 -6851.784,E2 -6851.784} C_VEL
LIN {X 0,Y 481.708,Z 167.482,A -85,B 0,C 180,E1 -6855.225,E2 -6855.225} C_VEL
LIN {X 0,Y 481.677,Z 167.486,A -85,B 0,C 180,E1 -6858.723,E2 -6858.723} C_VEL
LIN {X 0,Y 481.644,Z 167.492,A -85,B 0,C 180,E1 -6861.395,E2 -6861.395} C_VEL
LIN {X 0,Y 481.667,Z 167.485,A -85,B 0,C 180,E1 -6864.114,E2 -6864.114} C_VEL
LIN {X 0,Y 481.721,Z 167.481,A -85,B 0,C 180,E1 -6867.142,E2 -6867.142} C_VEL
LIN {X 0,Y 481.659,Z 167.486,A -85,B 0,C 180,E1 -6869.742,E2 -6869.742} C_VEL
LIN {X 0,Y 481.644,Z 167.49,A -85,B 0,C 180,E1 -6872.676,E2 -6872.676} C_VEL
LIN {X 0,Y 481.614,Z 167.494,A -85,B 0,C 180,E1 -6875.711,E2 -6875.711} C_VEL
LIN {X 0,Y 481.696,Z 167.483,A -85,B 0,C 180,E1 -6879.357,E2 -6879.357} C_VEL
LIN {X 0,Y 481.653,Z 167.488,A -85,B 0,C 180,E1 -6882.16,E2 -6882.16} C_VEL
LIN {X 0,Y 481.64,Z 167.492,A -85,B 0,C 180,E1 -6884.46,E2 -6884.46} C_VEL
LIN {X 0,Y 481.67,Z 167.488,A -85,B 0,C 180,E1 -6886.848,E2 -6886.848} C_VEL
LIN {X 0,Y 481.66,Z 167.492,A -85,B 0,C 180,E1 -6890.062,E2 -6890.062} C_VEL
LIN {X 0,Y 481.673,Z 167.542,A -85,B 0,C 180,E1 -6891.596,E2 -6891.596} C_VEL
LIN {X 0,Y 482.489,Z 173.198,A -85,B 0,C 180,E1 -6894.367,E2 -6894.367} C_VEL
LIN {X 0,Y 482.308,Z 178.687,A -85,B 0,C 180,E1 -6896.881,E2 -6896.881} C_VEL
LIN {X 0,Y 482.12,Z 185.306,A -85,B 0,C 180,E1 -6899.81,E2 -6899.81} C_VEL
LIN {X 0,Y 481.776,Z 193.085,A -85,B 0,C 180,E1 -6903.117,E2 -6903.117} C_VEL
LIN {X 0,Y 481.56,Z 199.768,A -85,B 0,C 180,E1 -6905.883,E2 -6905.883} C_VEL
LIN {X 0,Y 481.408,Z 207.737,A -85,B 0,C 180,E1 -6909.12,E2 -6909.12} C_VEL
LIN {X 0,Y 481.176,Z 215.296,A -85,B 0,C 180,E1 -6912.14,E2 -6912.14} C_VEL
LIN {X 0,Y 481.054,Z 222.784,A -85,B 0,C 180,E1 -6915.08,E2 -6915.08} C_VEL
LIN {X 0,Y 483.146,Z 236.058,A -85,B 0,C 180,E1 -6915.483,E2 -6915.483} C_VEL
LIN {X 0,Y 483.737,Z 243.027,A -85,B 0,C 180,E1 -6915.756,E2 -6915.756} C_VEL
LIN {X 0,Y 483.302,Z 255.436,A -85,B 0,C 180,E1 -6916.333,E2 -6916.333} C_VEL
LIN {X 0,Y 482.822,Z 267.915,A -85,B 0,C 180,E1 -6917.111,E2 -6917.111} C_VEL
LIN {X 0,Y 482.403,Z 279.367,A -85,B 0,C 180,E1 -6918.035,E2 -6918.035} C_VEL
LIN {X 0,Y 481.992,Z 289.711,A -85,B 0,C 180,E1 -6919.075,E2 -6919.075} C_VEL
LIN {X 0,Y 481.609,Z 298.216,A -85,B 0,C 180,E1 -6920.128,E2 -6920.128} C_VEL
LIN {X 0,Y 481.32,Z 306.511,A -85,B 0,C 180,E1 -6921.394,E2 -6921.394} C_VEL
LIN {X 0,Y 481.1,Z 313.195,A -85,B 0,C 180,E1 -6922.657,E2 -6922.657} C_VEL
LIN {X 0,Y 480.931,Z 319.311,A -85,B 0,C 180,E1 -6924.13,E2 -6924.13} C_VEL
LIN {X 0,Y 480.838,Z 323.283,A -85,B 0,C 180,E1 -6925.39,E2 -6925.39} C_VEL
LIN {X 0,Y 480.888,Z 326.219,A -85,B 0,C 180,E1 -6926.649,E2 -6926.649} C_VEL
LIN {X 0,Y 480.792,Z 328.609,A -85,B 0,C 180,E1 -6928.325,E2 -6928.325} C_VEL
LIN {X 0,Y 480.744,Z 329.432,A -85,B 0,C 180,E1 -6930.001,E2 -6930.001} C_VEL
LIN {X 0,Y 480.792,Z 328.611,A -85,B 0,C 180,E1 -6931.676,E2 -6931.676} C_VEL
LIN {X 0,Y 480.888,Z 326.224,A -85,B 0,C 180,E1 -6933.352,E2 -6933.352} C_VEL
LIN {X 0,Y 480.838,Z 323.289,A -85,B 0,C 180,E1 -6934.611,E2 -6934.611} C_VEL
LIN {X 0,Y 480.926,Z 319.321,A -85,B 0,C 180,E1 -6935.871,E2 -6935.871} C_VEL
LIN {X 0,Y 481.108,Z 313.221,A -85,B 0,C 180,E1 -6937.344,E2 -6937.344} C_VEL
LIN {X 0,Y 481.321,Z 306.556,A -85,B 0,C 180,E1 -6938.607,E2 -6938.607} C_VEL
LIN {X 0,Y 481.639,Z 298.288,A -85,B 0,C 180,E1 -6939.872,E2 -6939.872} C_VEL
LIN {X 0,Y 482.009,Z 289.823,A -85,B 0,C 180,E1 -6940.926,E2 -6940.926} C_VEL
LIN {X 0,Y 482.447,Z 279.394,A -85,B 0,C 180,E1 -6941.978,E2 -6941.978} C_VEL
LIN {X 0,Y 482.846,Z 268.321,A -85,B 0,C 180,E1 -6942.877,E2 -6942.877} C_VEL
LIN {X 0,Y 483.255,Z 257.708,A -85,B 0,C 180,E1 -6943.562,E2 -6943.562} C_VEL
LIN {X 0,Y 483.72,Z 246.154,A -85,B 0,C 180,E1 -6944.138,E2 -6944.138} C_VEL
LIN {X 0,Y 483.688,Z 239.797,A -85,B 0,C 180,E1 -6944.394,E2 -6944.394} C_VEL
LIN {X 0,Y 481.674,Z 226.359,A -85,B 0,C 180,E1 -6944.857,E2 -6944.857} C_VEL
LIN {X 0,Y 481.077,Z 222.612,A -85,B 0,C 180,E1 -6944.974,E2 -6944.974} C_VEL
LIN {X 0,Y 481.235,Z 214.176,A -85,B 0,C 180,E1 -6948.329,E2 -6948.329} C_VEL
LIN {X 0,Y 481.429,Z 206.604,A -85,B 0,C 180,E1 -6951.404,E2 -6951.404} C_VEL
LIN {X 0,Y 481.623,Z 198.867,A -85,B 0,C 180,E1 -6954.574,E2 -6954.574} C_VEL
LIN {X 0,Y 481.802,Z 192.737,A -85,B 0,C 180,E1 -6957.151,E2 -6957.151} C_VEL
LIN {X 0,Y 482.167,Z 185.692,A -85,B 0,C 180,E1 -6960.188,E2 -6960.188} C_VEL
LIN {X 0,Y 482.377,Z 179.156,A -85,B 0,C 180,E1 -6963.115,E2 -6963.115} C_VEL
LIN {X 0,Y 482.569,Z 173.768,A -85,B 0,C 180,E1 -6965.628,E2 -6965.628} C_VEL
LIN {X 0,Y 481.905,Z 168.925,A -85,B 0,C 180,E1 -6968.045,E2 -6968.045} C_VEL
LIN {X 0,Y 481.686,Z 167.49,A -85,B 0,C 180,E1 -6968.855,E2 -6968.855} C_VEL
LIN {X 0,Y 481.662,Z 167.489,A -85,B 0,C 180,E1 -6972.156,E2 -6972.156} C_VEL
LIN {X 0,Y 481.647,Z 167.487,A -85,B 0,C 180,E1 -6974.456,E2 -6974.456} C_VEL
LIN {X 0,Y 481.632,Z 167.491,A -85,B 0,C 180,E1 -6977.838,E2 -6977.838} C_VEL
LIN {X 0,Y 481.643,Z 167.49,A -85,B 0,C 180,E1 -6980.652,E2 -6980.652} C_VEL
LIN {X 0,Y 481.613,Z 167.495,A -85,B 0,C 180,E1 -6983.374,E2 -6983.374} C_VEL
LIN {X 0,Y 481.69,Z 167.481,A -85,B 0,C 180,E1 -6986.328,E2 -6986.328} C_VEL
LIN {X 0,Y 481.631,Z 167.491,A -85,B 0,C 180,E1 -6989.416,E2 -6989.416} C_VEL
LIN {X 0,Y 481.677,Z 167.486,A -85,B 0,C 180,E1 -6992.167,E2 -6992.167} C_VEL
LIN {X 0,Y 481.699,Z 167.483,A -85,B 0,C 180,E1 -6994.969,E2 -6994.969} C_VEL
LIN {X 0,Y 481.651,Z 167.486,A -85,B 0,C 180,E1 -6997.705,E2 -6997.705} C_VEL
LIN {X 0,Y 481.683,Z 167.485,A -85,B 0,C 180,E1 -7000.392,E2 -7000.392} C_VEL
LIN {X 0,Y 481.674,Z 167.485,A -85,B 0,C 180,E1 -7003.033,E2 -7003.033} C_VEL
LIN {X 0,Y 481.66,Z 167.488,A -85,B 0,C 180,E1 -7005.638,E2 -7005.638} C_VEL
LIN {X 0,Y 481.773,Z 167.473,A -85,B 0,C 180,E1 -7008.216,E2 -7008.216} C_VEL
LIN {X 0,Y 481.763,Z 167.472,A -85,B 0,C 180,E1 -7011.612,E2 -7011.612} C_VEL
LIN {X 0,Y 481.82,Z 167.471,A -85,B 0,C 180,E1 -7014.14,E2 -7014.14} C_VEL
LIN {X 0,Y 481.898,Z 167.458,A -85,B 0,C 180,E1 -7017.493,E2 -7017.493} C_VEL
LIN {X 0,Y 481.898,Z 167.458,A -85,B 0,C 180,E1 -7020.836,E2 -7020.836} C_VEL
LIN {X 0,Y 481.908,Z 167.457,A -85,B 0,C 180,E1 -7022.508,E2 -7022.508} C_VEL
LIN {X 0,Y 481.806,Z 167.473,A -85,B 0,C 180,E1 -7025.861,E2 -7025.861} C_VEL
LIN {X 0,Y 481.736,Z 167.478,A -85,B 0,C 180,E1 -7028.389,E2 -7028.389} C_VEL
LIN {X 0,Y 481.723,Z 167.48,A -85,B 0,C 180,E1 -7031.786,E2 -7031.786} C_VEL
LIN {X 0,Y 481.716,Z 167.479,A -85,B 0,C 180,E1 -7035.225,E2 -7035.225} C_VEL
LIN {X 0,Y 481.693,Z 167.482,A -85,B 0,C 180,E1 -7038.723,E2 -7038.723} C_VEL
LIN {X 0,Y 481.628,Z 167.492,A -85,B 0,C 180,E1 -7041.396,E2 -7041.396} C_VEL
LIN {X 0,Y 481.655,Z 167.489,A -85,B 0,C 180,E1 -7044.115,E2 -7044.115} C_VEL
LIN {X 0,Y 481.725,Z 167.48,A -85,B 0,C 180,E1 -7047.141,E2 -7047.141} C_VEL
LIN {X 0,Y 481.667,Z 167.485,A -85,B 0,C 180,E1 -7049.742,E2 -7049.742} C_VEL
LIN {X 0,Y 481.654,Z 167.49,A -85,B 0,C 180,E1 -7052.676,E2 -7052.676} C_VEL
LIN {X 0,Y 481.623,Z 167.493,A -85,B 0,C 180,E1 -7055.711,E2 -7055.711} C_VEL
LIN {X 0,Y 481.655,Z 167.488,A -85,B 0,C 180,E1 -7058.861,E2 -7058.861} C_VEL
LIN {X 0,Y 481.64,Z 167.487,A -85,B 0,C 180,E1 -7061.915,E2 -7061.915} C_VEL
LIN {X 0,Y 481.648,Z 167.491,A -85,B 0,C 180,E1 -7064.459,E2 -7064.459} C_VEL
LIN {X 0,Y 481.638,Z 167.491,A -85,B 0,C 180,E1 -7067.841,E2 -7067.841} C_VEL
LIN {X 0,Y 481.641,Z 167.491,A -85,B 0,C 180,E1 -7070.658,E2 -7070.658} C_VEL
LIN {X 0,Y 481.559,Z 167.501,A -85,B 0,C 180,E1 -7072.199,E2 -7072.199} C_VEL
LIN {X 0,Y 481.537,Z 168.739,A -85,B 0,C 180,E1 -7073.391,E2 -7073.391} C_VEL
LIN {X 0,Y 481.525,Z 172.854,A -85,B 0,C 180,E1 -7076.318,E2 -7076.318} C_VEL
LIN {X 0,Y 481.386,Z 177.399,A -85,B 0,C 180,E1 -7079.472,E2 -7079.472} C_VEL
LIN {X 0,Y 481.301,Z 181.342,A -85,B 0,C 180,E1 -7082.145,E2 -7082.145} C_VEL
LIN {X 0,Y 481.211,Z 185.55,A -85,B 0,C 180,E1 -7084.943,E2 -7084.943} C_VEL
LIN {X 0,Y 481.075,Z 189.831,A -85,B 0,C 180,E1 -7087.714,E2 -7087.714} C_VEL
LIN {X 0,Y 480.363,Z 190.981,A -85,B 0,C 180,E1 -7088.399,E2 -7088.399} C_VEL
LIN {X 0,Y 477.474,Z 193.001,A -85,B 0,C 180,E1 -7089.508,E2 -7089.508} C_VEL
LIN {X 0,Y 475.057,Z 194.629,A -85,B 0,C 180,E1 -7090.402,E2 -7090.402} C_VEL
LIN {X 0,Y 474.027,Z 195.815,A -85,B 0,C 180,E1 -7091.094,E2 -7091.094} C_VEL
LIN {X 0,Y 473.945,Z 196.191,A -85,B 0,C 180,E1 -7091.329,E2 -7091.329} C_VEL
LIN {X 0,Y 473.884,Z 198.645,A -85,B 0,C 180,E1 -7092.866,E2 -7092.866} C_VEL
LIN {X 0,Y 476.973,Z 213.668,A -85,B 0,C 180,E1 -7093.424,E2 -7093.424} C_VEL
LIN {X 0,Y 477.016,Z 221.331,A -85,B 0,C 180,E1 -7093.744,E2 -7093.744} C_VEL
LIN {X 0,Y 476.615,Z 233.528,A -85,B 0,C 180,E1 -7094.39,E2 -7094.39} C_VEL
LIN {X 0,Y 476.09,Z 244.494,A -85,B 0,C 180,E1 -7095.139,E2 -7095.139} C_VEL
LIN {X 0,Y 475.699,Z 254.559,A -85,B 0,C 180,E1 -7096,E2 -7096} C_VEL
LIN {X 0,Y 475.277,Z 263.794,A -85,B 0,C 180,E1 -7096.968,E2 -7096.968} C_VEL
LIN {X 0,Y 474.85,Z 272.202,A -85,B 0,C 180,E1 -7098.042,E2 -7098.042} C_VEL
LIN {X 0,Y 474.501,Z 280.402,A -85,B 0,C 180,E1 -7099.331,E2 -7099.331} C_VEL
LIN {X 0,Y 474.219,Z 286.994,A -85,B 0,C 180,E1 -7100.618,E2 -7100.618} C_VEL
LIN {X 0,Y 474.037,Z 292.24,A -85,B 0,C 180,E1 -7101.903,E2 -7101.903} C_VEL
LIN {X 0,Y 473.895,Z 296.316,A -85,B 0,C 180,E1 -7103.186,E2 -7103.186} C_VEL
LIN {X 0,Y 473.84,Z 298.451,A -85,B 0,C 180,E1 -7104.04,E2 -7104.04} C_VEL
LIN {X 0,Y 473.778,Z 300.124,A -85,B 0,C 180,E1 -7104.894,E2 -7104.894} C_VEL
LIN {X 0,Y 473.807,Z 302.277,A -85,B 0,C 180,E1 -7106.598,E2 -7106.598} C_VEL
LIN {X 0,Y 473.74,Z 302.74,A -85,B 0,C 180,E1 -7107.449,E2 -7107.449} C_VEL
LIN {X 0,Y 473.691,Z 302.481,A -85,B 0,C 180,E1 -7109.149,E2 -7109.149} C_VEL
LIN {X 0,Y 473.675,Z 301.783,A -85,B 0,C 180,E1 -7109.999,E2 -7109.999} C_VEL
LIN {X 0,Y 473.697,Z 300.67,A -85,B 0,C 180,E1 -7110.849,E2 -7110.849} C_VEL
LIN {X 0,Y 473.786,Z 299.127,A -85,B 0,C 180,E1 -7111.699,E2 -7111.699} C_VEL
LIN {X 0,Y 473.955,Z 296.034,A -85,B 0,C 180,E1 -7112.974,E2 -7112.974} C_VEL
LIN {X 0,Y 474.074,Z 291.899,A -85,B 0,C 180,E1 -7114.25,E2 -7114.25} C_VEL
LIN {X 0,Y 474.227,Z 285.602,A -85,B 0,C 180,E1 -7115.74,E2 -7115.74} C_VEL
LIN {X 0,Y 474.615,Z 279.329,A -85,B 0,C 180,E1 -7116.913,E2 -7116.913} C_VEL
LIN {X 0,Y 474.842,Z 271.734,A -85,B 0,C 180,E1 -7118.082,E2 -7118.082} C_VEL
LIN {X 0,Y 475.29,Z 263.269,A -85,B 0,C 180,E1 -7119.145,E2 -7119.145} C_VEL
LIN {X 0,Y 475.767,Z 252.823,A -85,B 0,C 180,E1 -7120.209,E2 -7120.209} C_VEL
LIN {X 0,Y 476.12,Z 242.479,A -85,B 0,C 180,E1 -7121.062,E2 -7121.062} C_VEL
LIN {X 0,Y 476.564,Z 231.115,A -85,B 0,C 180,E1 -7121.806,E2 -7121.806} C_VEL
LIN {X 0,Y 477.016,Z 218.536,A -85,B 0,C 180,E1 -7122.422,E2 -7122.422} C_VEL
LIN {X 0,Y 476.911,Z 213.323,A -85,B 0,C 180,E1 -7122.633,E2 -7122.633} C_VEL
LIN {X 0,Y 474.076,Z 199.781,A -85,B 0,C 180,E1 -7123.122,E2 -7123.122} C_VEL
LIN {X 0,Y 473.894,Z 198.581,A -85,B 0,C 180,E1 -7123.195,E2 -7123.195} C_VEL
LIN {X 0,Y 473.997,Z 194.907,A -85,B 0,C 180,E1 -7125.477,E2 -7125.477} C_VEL
LIN {X 0,Y 474.026,Z 189.287,A -85,B 0,C 180,E1 -7129.035,E2 -7129.035} C_VEL
LIN {X 0,Y 474.133,Z 185.14,A -85,B 0,C 180,E1 -7131.749,E2 -7131.749} C_VEL
LIN {X 0,Y 474.222,Z 181.01,A -85,B 0,C 180,E1 -7134.514,E2 -7134.514} C_VEL
LIN {X 0,Y 474.312,Z 176.844,A -85,B 0,C 180,E1 -7137.341,E2 -7137.341} C_VEL
LIN {X 0,Y 474.423,Z 172.664,A -85,B 0,C 180,E1 -7140.24,E2 -7140.24} C_VEL
LIN {X 0,Y 474.464,Z 168.465,A -85,B 0,C 180,E1 -7143.231,E2 -7143.231} C_VEL
LIN {X 0,Y 474.595,Z 168.368,A -85,B 0,C 180,E1 -7145.465,E2 -7145.465} C_VEL
LIN {X 0,Y 474.596,Z 168.368,A -85,B 0,C 180,E1 -7148.455,E2 -7148.455} C_VEL
LIN {X 0,Y 474.614,Z 168.368,A -85,B 0,C 180,E1 -7151.782,E2 -7151.782} C_VEL
LIN {X 0,Y 474.604,Z 168.365,A -85,B 0,C 180,E1 -7154.7,E2 -7154.7} C_VEL
LIN {X 0,Y 474.63,Z 168.361,A -85,B 0,C 180,E1 -7157.757,E2 -7157.757} C_VEL
LIN {X 0,Y 474.647,Z 168.361,A -85,B 0,C 180,E1 -7160.454,E2 -7160.454} C_VEL
LIN {X 0,Y 474.565,Z 168.372,A -85,B 0,C 180,E1 -7163.674,E2 -7163.674} C_VEL
LIN {X 0,Y 474.617,Z 168.364,A -85,B 0,C 180,E1 -7166.777,E2 -7166.777} C_VEL
LIN {X 0,Y 474.586,Z 168.368,A -85,B 0,C 180,E1 -7169.768,E2 -7169.768} C_VEL
LIN {X 0,Y 474.686,Z 168.358,A -85,B 0,C 180,E1 -7172.679,E2 -7172.679} C_VEL
LIN {X 0,Y 474.647,Z 168.358,A -85,B 0,C 180,E1 -7175.506,E2 -7175.506} C_VEL
LIN {X 0,Y 474.643,Z 168.361,A -85,B 0,C 180,E1 -7179.184,E2 -7179.184} C_VEL
LIN {X 0,Y 474.623,Z 168.366,A -85,B 0,C 180,E1 -7181.883,E2 -7181.883} C_VEL
LIN {X 0,Y 474.666,Z 168.359,A -85,B 0,C 180,E1 -7184.543,E2 -7184.543} C_VEL
LIN {X 0,Y 474.713,Z 168.353,A -85,B 0,C 180,E1 -7188.038,E2 -7188.038} C_VEL
LIN {X 0,Y 474.721,Z 168.35,A -85,B 0,C 180,E1 -7191.486,E2 -7191.486} C_VEL
LIN {X 0,Y 474.773,Z 168.347,A -85,B 0,C 180,E1 -7194.052,E2 -7194.052} C_VEL
LIN {X 0,Y 474.857,Z 168.337,A -85,B 0,C 180,E1 -7197.455,E2 -7197.455} C_VEL
LIN {X 0,Y 474.839,Z 168.338,A -85,B 0,C 180,E1 -7200.848,E2 -7200.848} C_VEL
LIN {X 0,Y 474.866,Z 168.334,A -85,B 0,C 180,E1 -7202.545,E2 -7202.545} C_VEL
LIN {X 0,Y 474.767,Z 168.348,A -85,B 0,C 180,E1 -7205.948,E2 -7205.948} C_VEL
LIN {X 0,Y 474.721,Z 168.349,A -85,B 0,C 180,E1 -7208.514,E2 -7208.514} C_VEL
LIN {X 0,Y 474.708,Z 168.352,A -85,B 0,C 180,E1 -7211.962,E2 -7211.962} C_VEL
LIN {X 0,Y 474.664,Z 168.358,A -85,B 0,C 180,E1 -7215.457,E2 -7215.457} C_VEL
LIN {X 0,Y 474.63,Z 168.363,A -85,B 0,C 180,E1 -7219.012,E2 -7219.012} C_VEL
LIN {X 0,Y 474.612,Z 168.366,A -85,B 0,C 180,E1 -7221.728,E2 -7221.728} C_VEL
LIN {X 0,Y 474.645,Z 168.36,A -85,B 0,C 180,E1 -7224.494,E2 -7224.494} C_VEL
LIN {X 0,Y 474.669,Z 168.357,A -85,B 0,C 180,E1 -7227.341,E2 -7227.341} C_VEL
LIN {X 0,Y 474.581,Z 168.37,A -85,B 0,C 180,E1 -7230.813,E2 -7230.813} C_VEL
LIN {X 0,Y 474.611,Z 168.367,A -85,B 0,C 180,E1 -7233.986,E2 -7233.986} C_VEL
LIN {X 0,Y 474.549,Z 168.374,A -85,B 0,C 180,E1 -7236.902,E2 -7236.902} C_VEL
LIN {X 0,Y 474.631,Z 168.363,A -85,B 0,C 180,E1 -7239.654,E2 -7239.654} C_VEL
LIN {X 0,Y 474.631,Z 168.362,A -85,B 0,C 180,E1 -7242.933,E2 -7242.933} C_VEL
LIN {X 0,Y 474.599,Z 168.37,A -85,B 0,C 180,E1 -7245.899,E2 -7245.899} C_VEL
LIN {X 0,Y 474.616,Z 168.37,A -85,B 0,C 180,E1 -7249.043,E2 -7249.043} C_VEL
LIN {X 0,Y 474.663,Z 168.431,A -85,B 0,C 180,E1 -7251.416,E2 -7251.416} C_VEL
LIN {X 0,Y 475.478,Z 174.399,A -85,B 0,C 180,E1 -7254.385,E2 -7254.385} C_VEL
LIN {X 0,Y 475.311,Z 179.661,A -85,B 0,C 180,E1 -7256.836,E2 -7256.836} C_VEL
LIN {X 0,Y 475.1,Z 186.281,A -85,B 0,C 180,E1 -7259.808,E2 -7259.808} C_VEL
LIN {X 0,Y 474.719,Z 194.049,A -85,B 0,C 180,E1 -7263.16,E2 -7263.16} C_VEL
LIN {X 0,Y 474.502,Z 200.718,A -85,B 0,C 180,E1 -7265.966,E2 -7265.966} C_VEL
LIN {X 0,Y 474.328,Z 208.481,A -85,B 0,C 180,E1 -7269.172,E2 -7269.172} C_VEL
LIN {X 0,Y 474.094,Z 216.211,A -85,B 0,C 180,E1 -7272.31,E2 -7272.31} C_VEL
LIN {X 0,Y 473.998,Z 222.502,A -85,B 0,C 180,E1 -7274.853,E2 -7274.853} C_VEL
LIN {X 0,Y 476.159,Z 236.395,A -85,B 0,C 180,E1 -7275.292,E2 -7275.292} C_VEL
LIN {X 0,Y 476.831,Z 242.643,A -85,B 0,C 180,E1 -7275.545,E2 -7275.545} C_VEL
LIN {X 0,Y 476.4,Z 255.099,A -85,B 0,C 180,E1 -7276.131,E2 -7276.131} C_VEL
LIN {X 0,Y 475.912,Z 267.062,A -85,B 0,C 180,E1 -7276.879,E2 -7276.879} C_VEL
LIN {X 0,Y 475.506,Z 278.255,A -85,B 0,C 180,E1 -7277.782,E2 -7277.782} C_VEL
LIN {X 0,Y 475.088,Z 287.496,A -85,B 0,C 180,E1 -7278.698,E2 -7278.698} C_VEL
LIN {X 0,Y 474.617,Z 296.374,A -85,B 0,C 180,E1 -7279.766,E2 -7279.766} C_VEL
LIN {X 0,Y 474.304,Z 305.038,A -85,B 0,C 180,E1 -7281.051,E2 -7281.051} C_VEL
LIN {X 0,Y 474.032,Z 311.953,A -85,B 0,C 180,E1 -7282.333,E2 -7282.333} C_VEL
LIN {X 0,Y 473.902,Z 317.147,A -85,B 0,C 180,E1 -7283.523,E2 -7283.523} C_VEL
LIN {X 0,Y 473.83,Z 321.844,A -85,B 0,C 180,E1 -7284.895,E2 -7284.895} C_VEL
LIN {X 0,Y 473.733,Z 324.142,A -85,B 0,C 180,E1 -7285.747,E2 -7285.747} C_VEL
LIN {X 0,Y 473.795,Z 326.011,A -85,B 0,C 180,E1 -7286.599,E2 -7286.599} C_VEL
LIN {X 0,Y 473.741,Z 327.409,A -85,B 0,C 180,E1 -7287.45,E2 -7287.45} C_VEL
LIN {X 0,Y 473.688,Z 329.016,A -85,B 0,C 180,E1 -7289.151,E2 -7289.151} C_VEL
LIN {X 0,Y 473.67,Z 329.235,A -85,B 0,C 180,E1 -7290.001,E2 -7290.001} C_VEL
LIN {X 0,Y 473.688,Z 329.022,A -85,B 0,C 180,E1 -7290.851,E2 -7290.851} C_VEL
LIN {X 0,Y 473.741,Z 327.426,A -85,B 0,C 180,E1 -7292.551,E2 -7292.551} C_VEL
LIN {X 0,Y 473.795,Z 326.036,A -85,B 0,C 180,E1 -7293.402,E2 -7293.402} C_VEL
LIN {X 0,Y 473.762,Z 323.105,A -85,B 0,C 180,E1 -7294.68,E2 -7294.68} C_VEL
LIN {X 0,Y 473.834,Z 319.141,A -85,B 0,C 180,E1 -7295.96,E2 -7295.96} C_VEL
LIN {X 0,Y 474.019,Z 313.051,A -85,B 0,C 180,E1 -7297.454,E2 -7297.454} C_VEL
LIN {X 0,Y 474.283,Z 306.394,A -85,B 0,C 180,E1 -7298.736,E2 -7298.736} C_VEL
LIN {X 0,Y 474.582,Z 298.135,A -85,B 0,C 180,E1 -7300.021,E2 -7300.021} C_VEL
LIN {X 0,Y 475.03,Z 289.685,A -85,B 0,C 180,E1 -7301.089,E2 -7301.089} C_VEL
LIN {X 0,Y 475.473,Z 279.471,A -85,B 0,C 180,E1 -7302.138,E2 -7302.138} C_VEL
LIN {X 0,Y 475.929,Z 267.932,A -85,B 0,C 180,E1 -7303.09,E2 -7303.09} C_VEL
LIN {X 0,Y 476.447,Z 255.756,A -85,B 0,C 180,E1 -7303.868,E2 -7303.868} C_VEL
LIN {X 0,Y 476.898,Z 243.548,A -85,B 0,C 180,E1 -7304.454,E2 -7304.454} C_VEL
LIN {X 0,Y 475.821,Z 233.414,A -85,B 0,C 180,E1 -7304.856,E2 -7304.856} C_VEL
LIN {X 0,Y 474.011,Z 222.44,A -85,B 0,C 180,E1 -7305.203,E2 -7305.203} C_VEL
LIN {X 0,Y 474.161,Z 214.431,A -85,B 0,C 180,E1 -7308.449,E2 -7308.449} C_VEL
LIN {X 0,Y 474.389,Z 206.481,A -85,B 0,C 180,E1 -7311.737,E2 -7311.737} C_VEL
LIN {X 0,Y 474.624,Z 198.772,A -85,B 0,C 180,E1 -7314.958,E2 -7314.958} C_VEL
LIN {X 0,Y 474.9,Z 191.073,A -85,B 0,C 180,E1 -7318.264,E2 -7318.264} C_VEL
LIN {X 0,Y 475.168,Z 185.084,A -85,B 0,C 180,E1 -7320.924,E2 -7320.924} C_VEL
LIN {X 0,Y 475.471,Z 178.105,A -85,B 0,C 180,E1 -7324.132,E2 -7324.132} C_VEL
LIN {X 0,Y 475.454,Z 173.731,A -85,B 0,C 180,E1 -7326.245,E2 -7326.245} C_VEL
LIN {X 0,Y 474.652,Z 168.366,A -85,B 0,C 180,E1 -7329.063,E2 -7329.063} C_VEL
LIN {X 0,Y 474.637,Z 168.363,A -85,B 0,C 180,E1 -7332.238,E2 -7332.238} C_VEL
LIN {X 0,Y 474.607,Z 168.368,A -85,B 0,C 180,E1 -7335.295,E2 -7335.295} C_VEL
LIN {X 0,Y 474.604,Z 168.368,A -85,B 0,C 180,E1 -7338.213,E2 -7338.213} C_VEL
LIN {X 0,Y 474.594,Z 168.369,A -85,B 0,C 180,E1 -7341.541,E2 -7341.541} C_VEL
LIN {X 0,Y 474.611,Z 168.363,A -85,B 0,C 180,E1 -7344.725,E2 -7344.725} C_VEL
LIN {X 0,Y 474.616,Z 168.364,A -85,B 0,C 180,E1 -7347.786,E2 -7347.786} C_VEL
LIN {X 0,Y 474.603,Z 168.368,A -85,B 0,C 180,E1 -7350.883,E2 -7350.883} C_VEL
LIN {X 0,Y 474.638,Z 168.364,A -85,B 0,C 180,E1 -7353.627,E2 -7353.627} C_VEL
LIN {X 0,Y 474.63,Z 168.363,A -85,B 0,C 180,E1 -7356.635,E2 -7356.635} C_VEL
LIN {X 0,Y 474.651,Z 168.361,A -85,B 0,C 180,E1 -7359.185,E2 -7359.185} C_VEL
LIN {X 0,Y 474.645,Z 168.361,A -85,B 0,C 180,E1 -7361.884,E2 -7361.884} C_VEL
LIN {X 0,Y 474.673,Z 168.358,A -85,B 0,C 180,E1 -7364.544,E2 -7364.544} C_VEL
LIN {X 0,Y 474.716,Z 168.352,A -85,B 0,C 180,E1 -7368.038,E2 -7368.038} C_VEL
LIN {X 0,Y 474.722,Z 168.349,A -85,B 0,C 180,E1 -7371.487,E2 -7371.487} C_VEL
LIN {X 0,Y 474.782,Z 168.346,A -85,B 0,C 180,E1 -7374.053,E2 -7374.053} C_VEL
LIN {X 0,Y 474.865,Z 168.334,A -85,B 0,C 180,E1 -7377.455,E2 -7377.455} C_VEL
LIN {X 0,Y 474.849,Z 168.336,A -85,B 0,C 180,E1 -7380.848,E2 -7380.848} C_VEL
LIN {X 0,Y 474.875,Z 168.333,A -85,B 0,C 180,E1 -7382.545,E2 -7382.545} C_VEL
LIN {X 0,Y 474.766,Z 168.349,A -85,B 0,C 180,E1 -7385.948,E2 -7385.948} C_VEL
LIN {X 0,Y 474.701,Z 168.355,A -85,B 0,C 180,E1 -7388.514,E2 -7388.514} C_VEL
LIN {X 0,Y 474.677,Z 168.358,A -85,B 0,C 180,E1 -7391.963,E2 -7391.963} C_VEL
LIN {X 0,Y 474.677,Z 168.361,A -85,B 0,C 180,E1 -7395.778,E2 -7395.778} C_VEL
LIN {X 0,Y 474.644,Z 168.361,A -85,B 0,C 180,E1 -7399.011,E2 -7399.011} C_VEL
LIN {X 0,Y 474.571,Z 168.37,A -85,B 0,C 180,E1 -7401.73,E2 -7401.73} C_VEL
LIN {X 0,Y 474.636,Z 168.362,A -85,B 0,C 180,E1 -7404.494,E2 -7404.494} C_VEL
LIN {X 0,Y 474.66,Z 168.361,A -85,B 0,C 180,E1 -7407.336,E2 -7407.336} C_VEL
LIN {X 0,Y 474.593,Z 168.365,A -85,B 0,C 180,E1 -7410.231,E2 -7410.231} C_VEL
LIN {X 0,Y 474.625,Z 168.364,A -85,B 0,C 180,E1 -7413.222,E2 -7413.222} C_VEL
LIN {X 0,Y 474.574,Z 168.371,A -85,B 0,C 180,E1 -7416.325,E2 -7416.325} C_VEL
LIN {X 0,Y 474.603,Z 168.366,A -85,B 0,C 180,E1 -7419.648,E2 -7419.648} C_VEL
LIN {X 0,Y 474.602,Z 168.368,A -85,B 0,C 180,E1 -7422.936,E2 -7422.936} C_VEL
LIN {X 0,Y 474.597,Z 168.367,A -85,B 0,C 180,E1 -7425.897,E2 -7425.897} C_VEL
LIN {X 0,Y 474.619,Z 168.366,A -85,B 0,C 180,E1 -7429.043,E2 -7429.043} C_VEL
LIN {X 0,Y 474.566,Z 168.373,A -85,B 0,C 180,E1 -7431.712,E2 -7431.712} C_VEL
LIN {X 0,Y 474.491,Z 168.604,A -85,B 0,C 180,E1 -7432.61,E2 -7432.61} C_VEL
LIN {X 0,Y 474.516,Z 171.472,A -85,B 0,C 180,E1 -7434.719,E2 -7434.719} C_VEL
LIN {X 0,Y 474.396,Z 175.772,A -85,B 0,C 180,E1 -7437.771,E2 -7437.771} C_VEL
LIN {X 0,Y 474.28,Z 180.358,A -85,B 0,C 180,E1 -7440.96,E2 -7440.96} C_VEL
LIN {X 0,Y 474.132,Z 184.249,A -85,B 0,C 180,E1 -7443.598,E2 -7443.598} C_VEL
LIN {X 0,Y 474.082,Z 189.071,A -85,B 0,C 180,E1 -7446.798,E2 -7446.798} C_VEL
LIN {X 0,Y 473.946,Z 194.176,A -85,B 0,C 180,E1 -7450.059,E2 -7450.059} C_VEL
LIN {X 0,Y 473.945,Z 196.191,A -85,B 0,C 180,E1 -7451.329,E2 -7451.329} C_VEL
LIN {X 0,Y 473.785,Z 197.52,A -85,B 0,C 180,E1 -7451.757,E2 -7451.757} C_VEL
LIN {X 0,Y 473.268,Z 200.422,A -85,B 0,C 180,E1 -7452.213,E2 -7452.213} C_VEL
LIN {X 0,Y 472.558,Z 204.173,A -85,B 0,C 180,E1 -7452.582,E2 -7452.582} C_VEL
LIN {X 0,Y 471.589,Z 209.522,A -85,B 0,C 180,E1 -7452.937,E2 -7452.937} C_VEL
LIN {X 0,Y 470.182,Z 221.204,A -85,B 0,C 180,E1 -7453.507,E2 -7453.507} C_VEL
LIN {X 0,Y 469.827,Z 231.912,A -85,B 0,C 180,E1 -7454.066,E2 -7454.066} C_VEL
LIN {X 0,Y 469.275,Z 242.986,A -85,B 0,C 180,E1 -7454.807,E2 -7454.807} C_VEL
LIN {X 0,Y 468.831,Z 253.353,A -85,B 0,C 180,E1 -7455.68,E2 -7455.68} C_VEL
LIN {X 0,Y 468.321,Z 263.81,A -85,B 0,C 180,E1 -7456.771,E2 -7456.771} C_VEL
LIN {X 0,Y 467.824,Z 272.253,A -85,B 0,C 180,E1 -7457.859,E2 -7457.859} C_VEL
LIN {X 0,Y 467.513,Z 280.477,A -85,B 0,C 180,E1 -7459.169,E2 -7459.169} C_VEL
LIN {X 0,Y 467.196,Z 287.091,A -85,B 0,C 180,E1 -7460.475,E2 -7460.475} C_VEL
LIN {X 0,Y 466.987,Z 292.356,A -85,B 0,C 180,E1 -7461.78,E2 -7461.78} C_VEL
LIN {X 0,Y 466.827,Z 296.451,A -85,B 0,C 180,E1 -7463.083,E2 -7463.083} C_VEL
LIN {X 0,Y 466.757,Z 298.604,A -85,B 0,C 180,E1 -7463.95,E2 -7463.95} C_VEL
LIN {X 0,Y 466.711,Z 300.284,A -85,B 0,C 180,E1 -7464.816,E2 -7464.816} C_VEL
LIN {X 0,Y 466.716,Z 302.454,A -85,B 0,C 180,E1 -7466.546,E2 -7466.546} C_VEL
LIN {X 0,Y 466.661,Z 302.934,A -85,B 0,C 180,E1 -7467.41,E2 -7467.41} C_VEL
LIN {X 0,Y 466.621,Z 302.69,A -85,B 0,C 180,E1 -7469.136,E2 -7469.136} C_VEL
LIN {X 0,Y 466.604,Z 302,A -85,B 0,C 180,E1 -7469.999,E2 -7469.999} C_VEL
LIN {X 0,Y 466.628,Z 300.904,A -85,B 0,C 180,E1 -7470.862,E2 -7470.862} C_VEL
LIN {X 0,Y 466.721,Z 299.369,A -85,B 0,C 180,E1 -7471.725,E2 -7471.725} C_VEL
LIN {X 0,Y 466.868,Z 296.295,A -85,B 0,C 180,E1 -7473.019,E2 -7473.019} C_VEL
LIN {X 0,Y 467.011,Z 292.178,A -85,B 0,C 180,E1 -7474.314,E2 -7474.314} C_VEL
LIN {X 0,Y 467.17,Z 285.901,A -85,B 0,C 180,E1 -7475.827,E2 -7475.827} C_VEL
LIN {X 0,Y 467.589,Z 278.307,A -85,B 0,C 180,E1 -7477.248,E2 -7477.248} C_VEL
LIN {X 0,Y 467.905,Z 270.501,A -85,B 0,C 180,E1 -7478.42,E2 -7478.42} C_VEL
LIN {X 0,Y 468.374,Z 261.722,A -85,B 0,C 180,E1 -7479.499,E2 -7479.499} C_VEL
LIN {X 0,Y 468.865,Z 250.917,A -85,B 0,C 180,E1 -7480.579,E2 -7480.579} C_VEL
LIN {X 0,Y 469.346,Z 239.998,A -85,B 0,C 180,E1 -7481.442,E2 -7481.442} C_VEL
LIN {X 0,Y 469.819,Z 227.589,A -85,B 0,C 180,E1 -7482.207,E2 -7482.207} C_VEL
LIN {X 0,Y 470.199,Z 215.807,A -85,B 0,C 180,E1 -7482.751,E2 -7482.751} C_VEL
LIN {X 0,Y 467.697,Z 203.004,A -85,B 0,C 180,E1 -7483.25,E2 -7483.25} C_VEL
LIN {X 0,Y 466.828,Z 198.789,A -85,B 0,C 180,E1 -7483.401,E2 -7483.401} C_VEL
LIN {X 0,Y 466.91,Z 195.127,A -85,B 0,C 180,E1 -7485.718,E2 -7485.718} C_VEL
LIN {X 0,Y 466.955,Z 190.735,A -85,B 0,C 180,E1 -7488.522,E2 -7488.522} C_VEL
LIN {X 0,Y 467.075,Z 186.692,A -85,B 0,C 180,E1 -7491.167,E2 -7491.167} C_VEL
LIN {X 0,Y 467.124,Z 182.546,A -85,B 0,C 180,E1 -7493.965,E2 -7493.965} C_VEL
LIN {X 0,Y 467.219,Z 178.38,A -85,B 0,C 180,E1 -7496.822,E2 -7496.822} C_VEL
LIN {X 0,Y 467.353,Z 174.194,A -85,B 0,C 180,E1 -7499.749,E2 -7499.749} C_VEL
LIN {X 0,Y 467.409,Z 170.162,A -85,B 0,C 180,E1 -7502.645,E2 -7502.645} C_VEL
LIN {X 0,Y 467.462,Z 169.26,A -85,B 0,C 180,E1 -7503.795,E2 -7503.795} C_VEL
LIN {X 0,Y 467.537,Z 169.246,A -85,B 0,C 180,E1 -7505.887,E2 -7505.887} C_VEL
LIN {X 0,Y 467.545,Z 169.246,A -85,B 0,C 180,E1 -7509.144,E2 -7509.144} C_VEL
LIN {X 0,Y 467.573,Z 169.242,A -85,B 0,C 180,E1 -7512.557,E2 -7512.557} C_VEL
LIN {X 0,Y 467.553,Z 169.245,A -85,B 0,C 180,E1 -7515.05,E2 -7515.05} C_VEL
LIN {X 0,Y 467.606,Z 169.238,A -85,B 0,C 180,E1 -7517.441,E2 -7517.441} C_VEL
LIN {X 0,Y 467.593,Z 169.243,A -85,B 0,C 180,E1 -7520.856,E2 -7520.856} C_VEL
LIN {X 0,Y 467.536,Z 169.248,A -85,B 0,C 180,E1 -7524.258,E2 -7524.258} C_VEL
LIN {X 0,Y 467.556,Z 169.247,A -85,B 0,C 180,E1 -7527.318,E2 -7527.318} C_VEL
LIN {X 0,Y 467.551,Z 169.245,A -85,B 0,C 180,E1 -7530.663,E2 -7530.663} C_VEL
LIN {X 0,Y 467.6,Z 169.238,A -85,B 0,C 180,E1 -7533.198,E2 -7533.198} C_VEL
LIN {X 0,Y 467.563,Z 169.242,A -85,B 0,C 180,E1 -7536.056,E2 -7536.056} C_VEL
LIN {X 0,Y 467.609,Z 169.237,A -85,B 0,C 180,E1 -7538.856,E2 -7538.856} C_VEL
LIN {X 0,Y 467.598,Z 169.239,A -85,B 0,C 180,E1 -7541.601,E2 -7541.601} C_VEL
LIN {X 0,Y 467.621,Z 169.236,A -85,B 0,C 180,E1 -7544.304,E2 -7544.304} C_VEL
LIN {X 0,Y 467.669,Z 169.23,A -85,B 0,C 180,E1 -7547.855,E2 -7547.855} C_VEL
LIN {X 0,Y 467.669,Z 169.228,A -85,B 0,C 180,E1 -7551.357,E2 -7551.357} C_VEL
LIN {X 0,Y 467.736,Z 169.224,A -85,B 0,C 180,E1 -7553.962,E2 -7553.962} C_VEL
LIN {X 0,Y 467.823,Z 169.213,A -85,B 0,C 180,E1 -7557.417,E2 -7557.417} C_VEL
LIN {X 0,Y 467.791,Z 169.215,A -85,B 0,C 180,E1 -7560.861,E2 -7560.861} C_VEL
LIN {X 0,Y 467.832,Z 169.21,A -85,B 0,C 180,E1 -7562.583,E2 -7562.583} C_VEL
LIN {X 0,Y 467.729,Z 169.224,A -85,B 0,C 180,E1 -7566.037,E2 -7566.037} C_VEL
LIN {X 0,Y 467.668,Z 169.228,A -85,B 0,C 180,E1 -7568.643,E2 -7568.643} C_VEL
LIN {X 0,Y 467.658,Z 169.23,A -85,B 0,C 180,E1 -7572.381,E2 -7572.381} C_VEL
LIN {X 0,Y 467.613,Z 169.237,A -85,B 0,C 180,E1 -7575.886,E2 -7575.886} C_VEL
LIN {X 0,Y 467.589,Z 169.24,A -85,B 0,C 180,E1 -7579.309,E2 -7579.309} C_VEL
LIN {X 0,Y 467.545,Z 169.245,A -85,B 0,C 180,E1 -7582.073,E2 -7582.073} C_VEL
LIN {X 0,Y 467.591,Z 169.241,A -85,B 0,C 180,E1 -7584.888,E2 -7584.888} C_VEL
LIN {X 0,Y 467.599,Z 169.236,A -85,B 0,C 180,E1 -7587.77,E2 -7587.77} C_VEL
LIN {X 0,Y 467.543,Z 169.245,A -85,B 0,C 180,E1 -7591.048,E2 -7591.048} C_VEL
LIN {X 0,Y 467.562,Z 169.246,A -85,B 0,C 180,E1 -7594.245,E2 -7594.245} C_VEL
LIN {X 0,Y 467.525,Z 169.249,A -85,B 0,C 180,E1 -7597.189,E2 -7597.189} C_VEL
LIN {X 0,Y 467.575,Z 169.242,A -85,B 0,C 180,E1 -7600.265,E2 -7600.265} C_VEL
LIN {X 0,Y 467.598,Z 169.242,A -85,B 0,C 180,E1 -7602.574,E2 -7602.574} C_VEL
LIN {X 0,Y 467.555,Z 169.248,A -85,B 0,C 180,E1 -7606.179,E2 -7606.179} C_VEL
LIN {X 0,Y 467.566,Z 169.247,A -85,B 0,C 180,E1 -7608.725,E2 -7608.725} C_VEL
LIN {X 0,Y 467.631,Z 169.356,A -85,B 0,C 180,E1 -7611.247,E2 -7611.247} C_VEL
LIN {X 0,Y 468.446,Z 175.161,A -85,B 0,C 180,E1 -7614.193,E2 -7614.193} C_VEL
LIN {X 0,Y 468.327,Z 179.542,A -85,B 0,C 180,E1 -7616.276,E2 -7616.276} C_VEL
LIN {X 0,Y 468.07,Z 186.145,A -85,B 0,C 180,E1 -7619.306,E2 -7619.306} C_VEL
LIN {X 0,Y 467.733,Z 192.788,A -85,B 0,C 180,E1 -7622.241,E2 -7622.241} C_VEL
